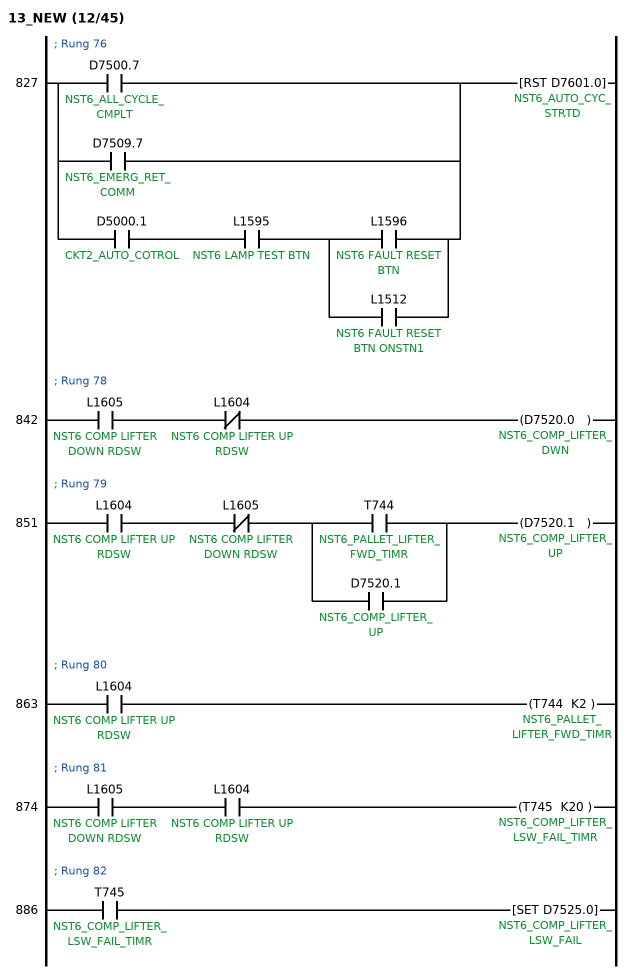
[picture p240: ladder of 13_NEW, rungs at steps 827 to 886]
; Rung 76
827   LD      D7500.7  ; NST6_ALL_CYCLE_CMPLT
      OR      D7509.7  ; NST6_EMERG_RET_COMM
      LD      D5000.1  ; CKT2_AUTO_COTROL
      AND     L1595  ; NST6 LAMP TEST BTN
      LD      L1596  ; NST6 FAULT RESET BTN
      OR      L1512  ; NST6 FAULT RESET BTN ONSTN1
      ANB
      ORB
      RST     D7601.0  ; NST6_AUTO_CYC_STRTD
; Rung 78
842   LD      L1605  ; NST6 COMP LIFTER DOWN RDSW
      ANI     L1604  ; NST6 COMP LIFTER UP RDSW
      OUT     D7520.0  ; NST6_COMP_LIFTER_DWN
; Rung 79
851   LD      L1604  ; NST6 COMP LIFTER UP RDSW
      ANI     L1605  ; NST6 COMP LIFTER DOWN RDSW
      LD      T744  ; NST6_PALLET_LIFTER_FWD_TIMR
      OR      D7520.1  ; NST6_COMP_LIFTER_UP
      ANB
      OUT     D7520.1  ; NST6_COMP_LIFTER_UP
; Rung 80
863   LD      L1604  ; NST6 COMP LIFTER UP RDSW
      OUT     T744 K2  ; NST6_PALLET_LIFTER_FWD_TIMR
; Rung 81
874   LD      L1605  ; NST6 COMP LIFTER DOWN RDSW
      AND     L1604  ; NST6 COMP LIFTER UP RDSW
      OUT     T745 K20  ; NST6_COMP_LIFTER_LSW_FAIL_TIMR
; Rung 82
886   LD      T745  ; NST6_COMP_LIFTER_LSW_FAIL_TIMR
      SET     D7525.0  ; NST6_COMP_LIFTER_LSW_FAIL
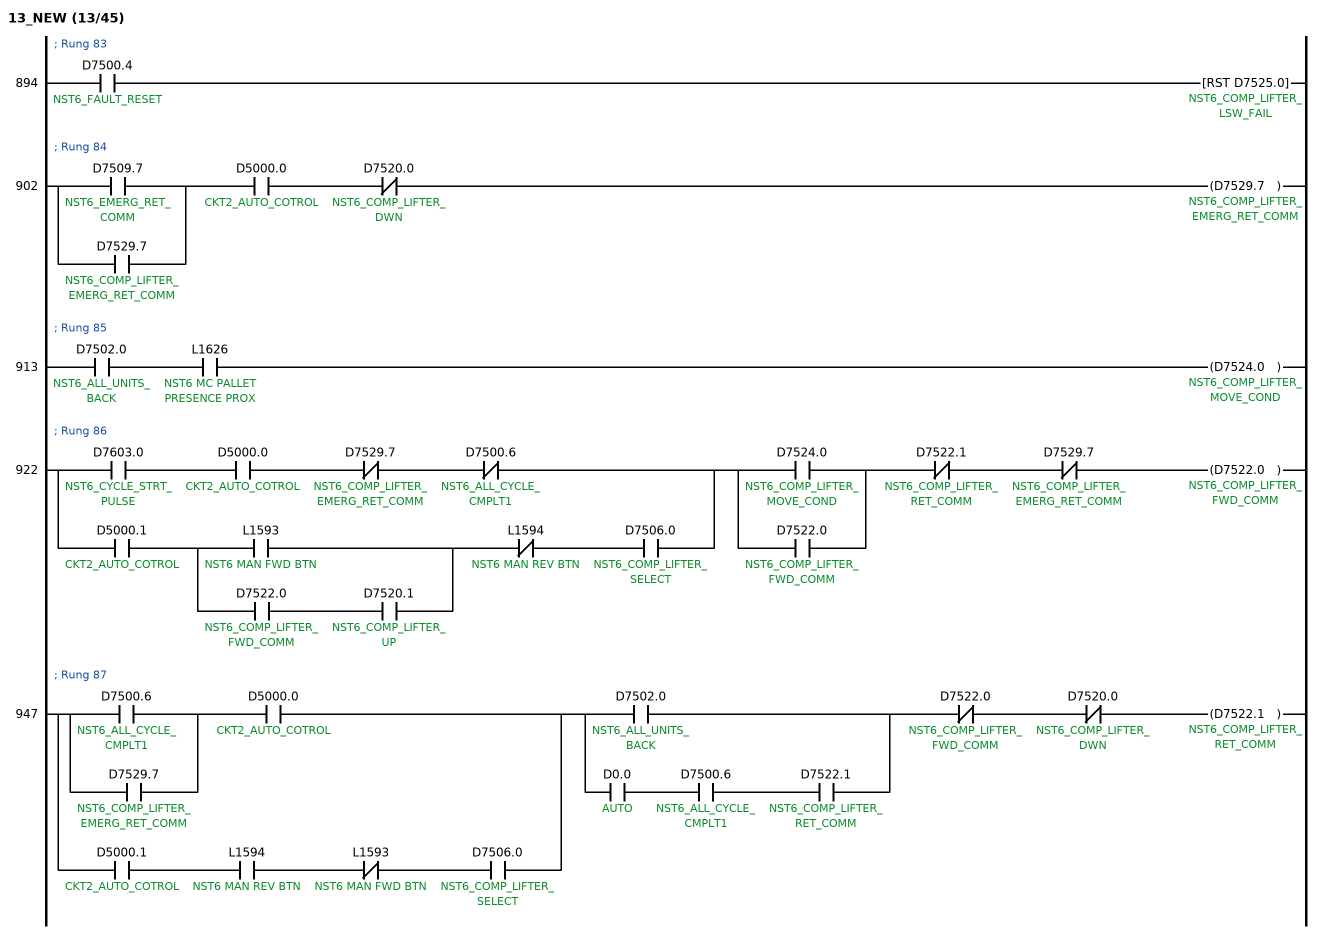
; Rung 83
894   LD      D7500.4  ; NST6_FAULT_RESET
      RST     D7525.0  ; NST6_COMP_LIFTER_LSW_FAIL
; Rung 84
902   LD      D7509.7  ; NST6_EMERG_RET_COMM
      OR      D7529.7  ; NST6_COMP_LIFTER_EMERG_RET_COMM
      AND     D5000.0  ; CKT2_AUTO_COTROL
      ANI     D7520.0  ; NST6_COMP_LIFTER_DWN
      OUT     D7529.7  ; NST6_COMP_LIFTER_EMERG_RET_COMM
; Rung 85
913   LD      D7502.0  ; NST6_ALL_UNITS_BACK
      AND     L1626  ; NST6 MC PALLET PRESENCE PROX
      OUT     D7524.0  ; NST6_COMP_LIFTER_MOVE_COND
; Rung 86
922   LD      D7603.0  ; NST6_CYCLE_STRT_PULSE
      AND     D5000.0  ; CKT2_AUTO_COTROL
      ANI     D7529.7  ; NST6_COMP_LIFTER_EMERG_RET_COMM
      ANI     D7500.6  ; NST6_ALL_CYCLE_CMPLT1
      LD      D5000.1  ; CKT2_AUTO_COTROL
      LD      L1593  ; NST6 MAN FWD BTN
      LD      D7522.0  ; NST6_COMP_LIFTER_FWD_COMM
      AND     D7520.1  ; NST6_COMP_LIFTER_UP
      ORB
      ANB
      ANI     L1594  ; NST6 MAN REV BTN
      AND     D7506.0  ; NST6_COMP_LIFTER_SELECT
      ORB
      LD      D7524.0  ; NST6_COMP_LIFTER_MOVE_COND
      OR      D7522.0  ; NST6_COMP_LIFTER_FWD_COMM
      ANB
      ANI     D7522.1  ; NST6_COMP_LIFTER_RET_COMM
      ANI     D7529.7  ; NST6_COMP_LIFTER_EMERG_RET_COMM
      OUT     D7522.0  ; NST6_COMP_LIFTER_FWD_COMM
; Rung 87
947   LD      D7500.6  ; NST6_ALL_CYCLE_CMPLT1
      OR      D7529.7  ; NST6_COMP_LIFTER_EMERG_RET_COMM
      AND     D5000.0  ; CKT2_AUTO_COTROL
      LD      D5000.1  ; CKT2_AUTO_COTROL
      AND     L1594  ; NST6 MAN REV BTN
      ANI     L1593  ; NST6 MAN FWD BTN
      AND     D7506.0  ; NST6_COMP_LIFTER_SELECT
      ORB
      LD      D7502.0  ; NST6_ALL_UNITS_BACK
      LD      D0.0  ; AUTO
      AND     D7500.6  ; NST6_ALL_CYCLE_CMPLT1
      AND     D7522.1  ; NST6_COMP_LIFTER_RET_COMM
      ORB
      ANB
      ANI     D7522.0  ; NST6_COMP_LIFTER_FWD_COMM
      ANI     D7520.0  ; NST6_COMP_LIFTER_DWN
      OUT     D7522.1  ; NST6_COMP_LIFTER_RET_COMM
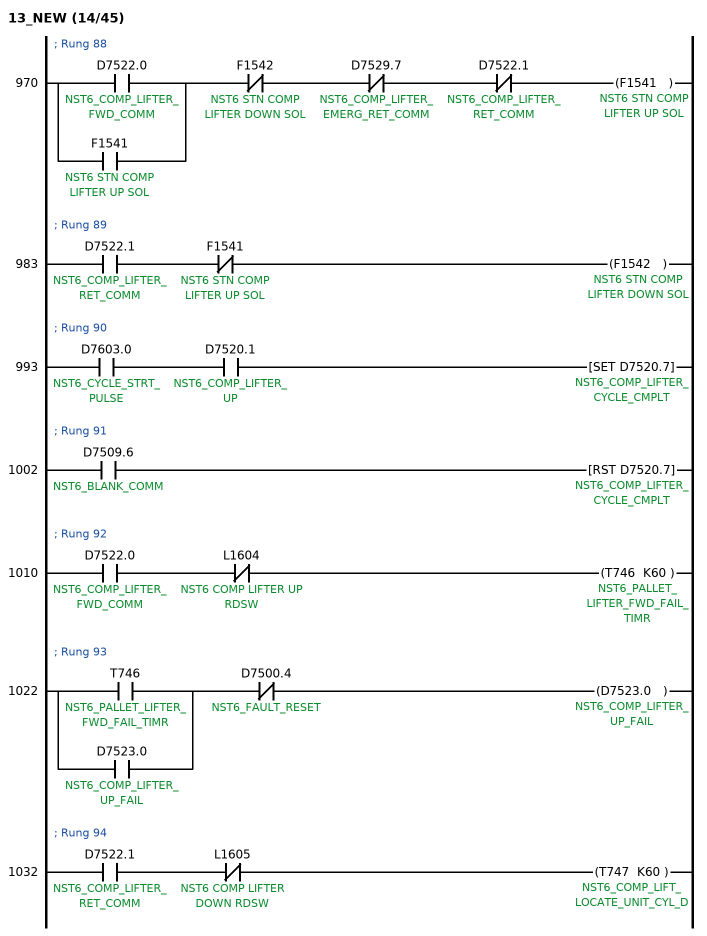
; Rung 88
970   LD      D7522.0  ; NST6_COMP_LIFTER_FWD_COMM
      OR      F1541  ; NST6 STN COMP LIFTER UP SOL
      ANI     F1542  ; NST6 STN COMP LIFTER DOWN SOL
      ANI     D7529.7  ; NST6_COMP_LIFTER_EMERG_RET_COMM
      ANI     D7522.1  ; NST6_COMP_LIFTER_RET_COMM
      OUT     F1541  ; NST6 STN COMP LIFTER UP SOL
; Rung 89
983   LD      D7522.1  ; NST6_COMP_LIFTER_RET_COMM
      ANI     F1541  ; NST6 STN COMP LIFTER UP SOL
      OUT     F1542  ; NST6 STN COMP LIFTER DOWN SOL
; Rung 90
993   LD      D7603.0  ; NST6_CYCLE_STRT_PULSE
      AND     D7520.1  ; NST6_COMP_LIFTER_UP
      SET     D7520.7  ; NST6_COMP_LIFTER_CYCLE_CMPLT
; Rung 91
1002  LD      D7509.6  ; NST6_BLANK_COMM
      RST     D7520.7  ; NST6_COMP_LIFTER_CYCLE_CMPLT
; Rung 92
1010  LD      D7522.0  ; NST6_COMP_LIFTER_FWD_COMM
      ANI     L1604  ; NST6 COMP LIFTER UP RDSW
      OUT     T746 K60  ; NST6_PALLET_LIFTER_FWD_FAIL_TIMR
; Rung 93
1022  LD      T746  ; NST6_PALLET_LIFTER_FWD_FAIL_TIMR
      OR      D7523.0  ; NST6_COMP_LIFTER_UP_FAIL
      ANI     D7500.4  ; NST6_FAULT_RESET
      OUT     D7523.0  ; NST6_COMP_LIFTER_UP_FAIL
; Rung 94
1032  LD      D7522.1  ; NST6_COMP_LIFTER_RET_COMM
      ANI     L1605  ; NST6 COMP LIFTER DOWN RDSW
      OUT     T747 K60  ; NST6_COMP_LIFT_LOCATE_UNIT_CYL_D
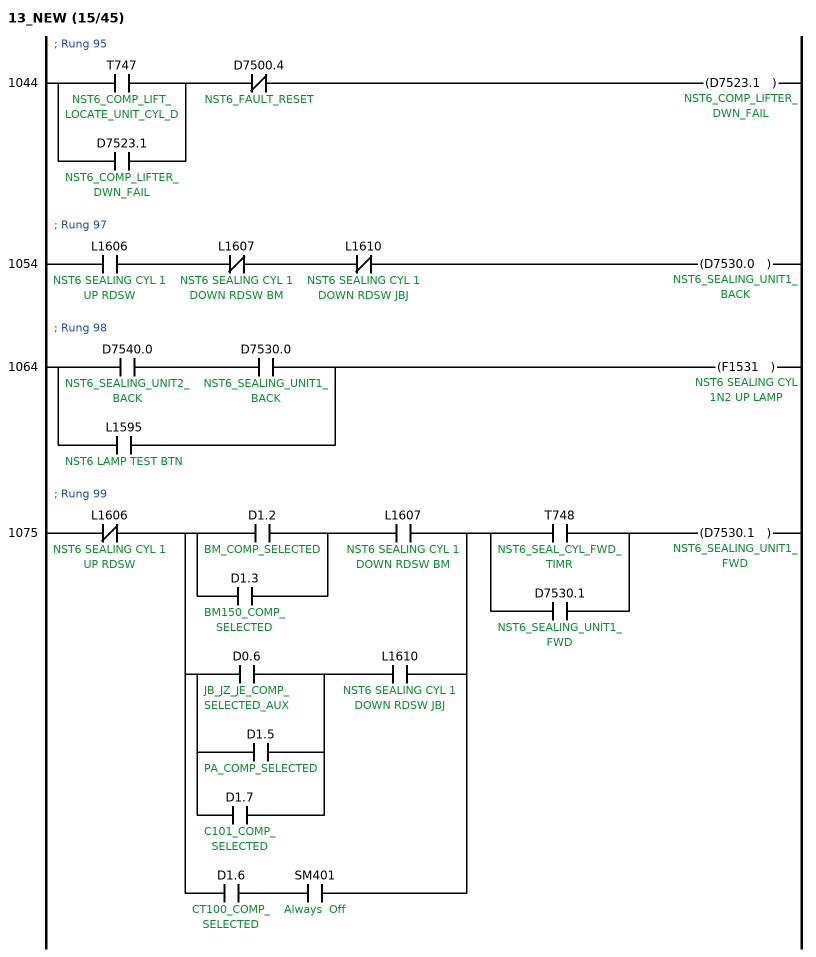
; Rung 95
1044  LD      T747  ; NST6_COMP_LIFT_LOCATE_UNIT_CYL_D
      OR      D7523.1  ; NST6_COMP_LIFTER_DWN_FAIL
      ANI     D7500.4  ; NST6_FAULT_RESET
      OUT     D7523.1  ; NST6_COMP_LIFTER_DWN_FAIL
; Rung 97
1054  LD      L1606  ; NST6 SEALING CYL 1 UP RDSW
      ANI     L1607  ; NST6 SEALING CYL 1 DOWN RDSW BM
      ANI     L1610  ; NST6 SEALING CYL 1 DOWN RDSW JBJ
      OUT     D7530.0  ; NST6_SEALING_UNIT1_BACK
; Rung 98
1064  LD      D7540.0  ; NST6_SEALING_UNIT2_BACK
      AND     D7530.0  ; NST6_SEALING_UNIT1_BACK
      OR      L1595  ; NST6 LAMP TEST BTN
      OUT     F1531  ; NST6 SEALING CYL 1N2 UP LAMP
; Rung 99
1075  LDI     L1606  ; NST6 SEALING CYL 1 UP RDSW
      LD      D1.2  ; BM_COMP_SELECTED
      OR      D1.3  ; BM150_COMP_SELECTED
      AND     L1607  ; NST6 SEALING CYL 1 DOWN RDSW BM
      LD      D0.6  ; JB_JZ_JE_COMP_SELECTED_AUX
      OR      D1.5  ; PA_COMP_SELECTED
      OR      D1.7  ; C101_COMP_SELECTED
      AND     L1610  ; NST6 SEALING CYL 1 DOWN RDSW JBJ
      ORB
      LD      D1.6  ; CT100_COMP_SELECTED
      AND     SM401  ; Always  Off
      ORB
      ANB
      LD      T748  ; NST6_SEAL_CYL_FWD_TIMR
      OR      D7530.1  ; NST6_SEALING_UNIT1_FWD
      ANB
      OUT     D7530.1  ; NST6_SEALING_UNIT1_FWD
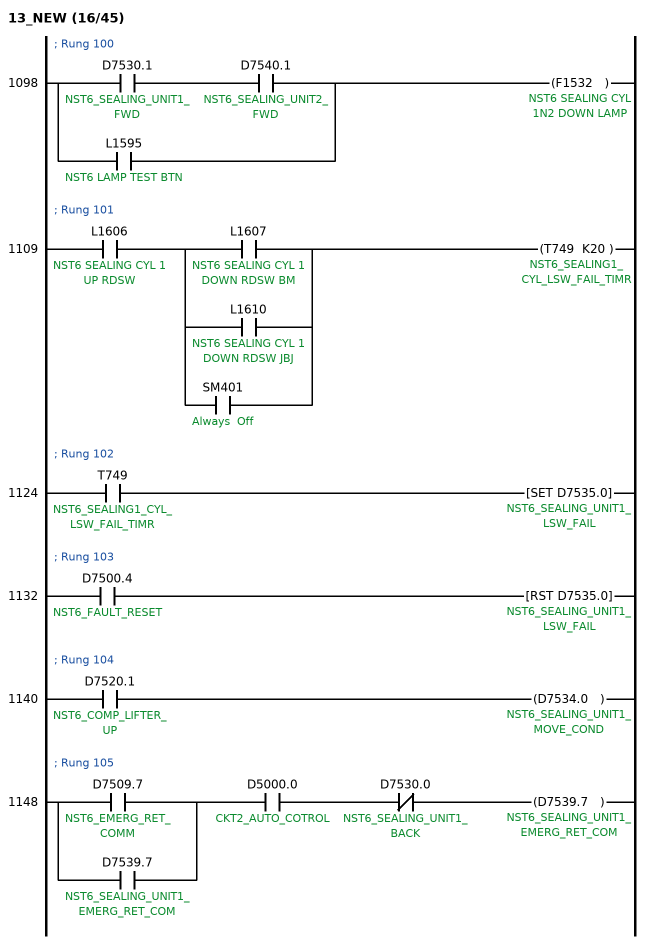
; Rung 100
1098  LD      D7530.1  ; NST6_SEALING_UNIT1_FWD
      AND     D7540.1  ; NST6_SEALING_UNIT2_FWD
      OR      L1595  ; NST6 LAMP TEST BTN
      OUT     F1532  ; NST6 SEALING CYL 1N2 DOWN LAMP
; Rung 101
1109  LD      L1606  ; NST6 SEALING CYL 1 UP RDSW
      LD      L1607  ; NST6 SEALING CYL 1 DOWN RDSW BM
      OR      L1610  ; NST6 SEALING CYL 1 DOWN RDSW JBJ
      OR      SM401  ; Always  Off
      ANB
      OUT     T749 K20  ; NST6_SEALING1_CYL_LSW_FAIL_TIMR
; Rung 102
1124  LD      T749  ; NST6_SEALING1_CYL_LSW_FAIL_TIMR
      SET     D7535.0  ; NST6_SEALING_UNIT1_LSW_FAIL
; Rung 103
1132  LD      D7500.4  ; NST6_FAULT_RESET
      RST     D7535.0  ; NST6_SEALING_UNIT1_LSW_FAIL
; Rung 104
1140  LD      D7520.1  ; NST6_COMP_LIFTER_UP
      OUT     D7534.0  ; NST6_SEALING_UNIT1_MOVE_COND
; Rung 105
1148  LD      D7509.7  ; NST6_EMERG_RET_COMM
      OR      D7539.7  ; NST6_SEALING_UNIT1_EMERG_RET_COM
      AND     D5000.0  ; CKT2_AUTO_COTROL
      ANI     D7530.0  ; NST6_SEALING_UNIT1_BACK
      OUT     D7539.7  ; NST6_SEALING_UNIT1_EMERG_RET_COM
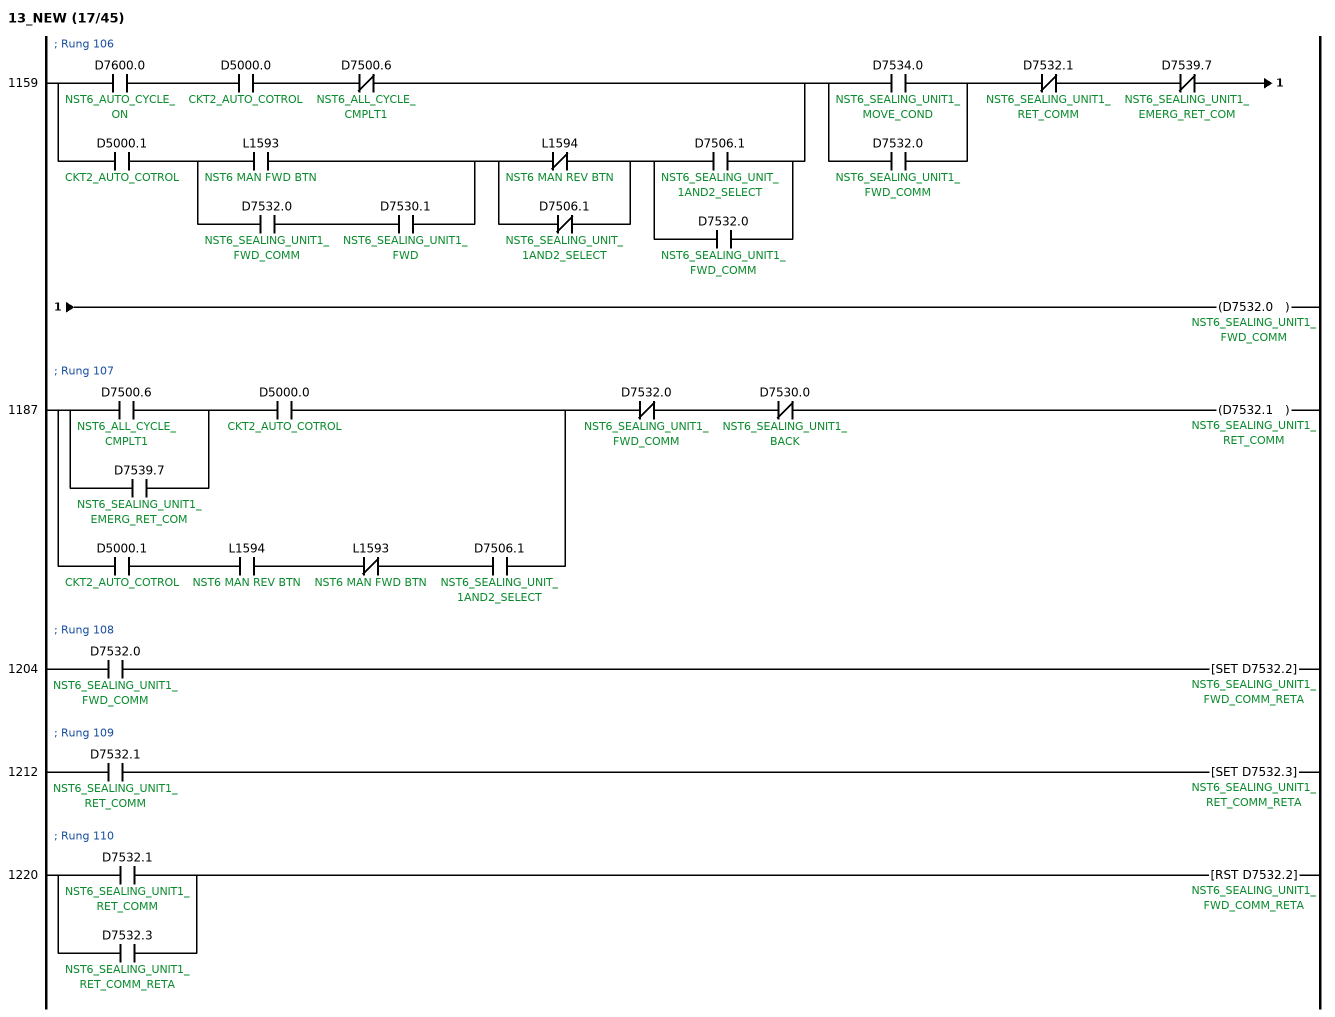
; Rung 106
1159  LD      D7600.0  ; NST6_AUTO_CYCLE_ON
      AND     D5000.0  ; CKT2_AUTO_COTROL
      ANI     D7500.6  ; NST6_ALL_CYCLE_CMPLT1
      LD      D5000.1  ; CKT2_AUTO_COTROL
      LD      L1593  ; NST6 MAN FWD BTN
      LD      D7532.0  ; NST6_SEALING_UNIT1_FWD_COMM
      AND     D7530.1  ; NST6_SEALING_UNIT1_FWD
      ORB
      ANB
      LDI     L1594  ; NST6 MAN REV BTN
      ORI     D7506.1  ; NST6_SEALING_UNIT_1AND2_SELECT
      ANB
      LD      D7506.1  ; NST6_SEALING_UNIT_1AND2_SELECT
      OR      D7532.0  ; NST6_SEALING_UNIT1_FWD_COMM
      ANB
      ORB
      LD      D7534.0  ; NST6_SEALING_UNIT1_MOVE_COND
      OR      D7532.0  ; NST6_SEALING_UNIT1_FWD_COMM
      ANB
      ANI     D7532.1  ; NST6_SEALING_UNIT1_RET_COMM
      ANI     D7539.7  ; NST6_SEALING_UNIT1_EMERG_RET_COM
      OUT     D7532.0  ; NST6_SEALING_UNIT1_FWD_COMM
; Rung 107
1187  LD      D7500.6  ; NST6_ALL_CYCLE_CMPLT1
      OR      D7539.7  ; NST6_SEALING_UNIT1_EMERG_RET_COM
      AND     D5000.0  ; CKT2_AUTO_COTROL
      LD      D5000.1  ; CKT2_AUTO_COTROL
      AND     L1594  ; NST6 MAN REV BTN
      ANI     L1593  ; NST6 MAN FWD BTN
      AND     D7506.1  ; NST6_SEALING_UNIT_1AND2_SELECT
      ORB
      ANI     D7532.0  ; NST6_SEALING_UNIT1_FWD_COMM
      ANI     D7530.0  ; NST6_SEALING_UNIT1_BACK
      OUT     D7532.1  ; NST6_SEALING_UNIT1_RET_COMM
; Rung 108
1204  LD      D7532.0  ; NST6_SEALING_UNIT1_FWD_COMM
      SET     D7532.2  ; NST6_SEALING_UNIT1_FWD_COMM_RETA
; Rung 109
1212  LD      D7532.1  ; NST6_SEALING_UNIT1_RET_COMM
      SET     D7532.3  ; NST6_SEALING_UNIT1_RET_COMM_RETA
; Rung 110
1220  LD      D7532.1  ; NST6_SEALING_UNIT1_RET_COMM
      OR      D7532.3  ; NST6_SEALING_UNIT1_RET_COMM_RETA
      RST     D7532.2  ; NST6_SEALING_UNIT1_FWD_COMM_RETA
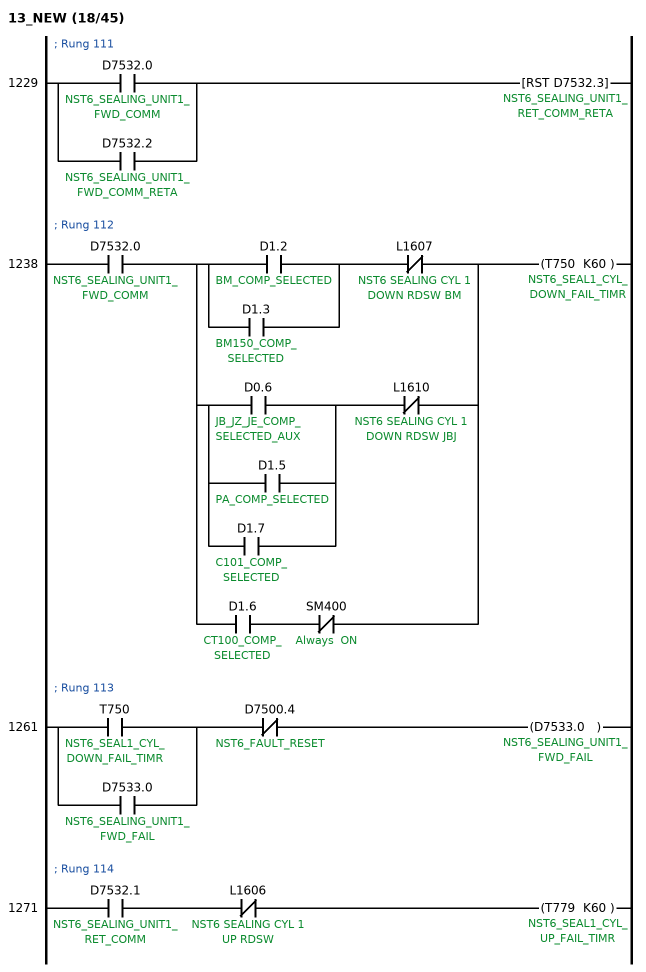
; Rung 111
1229  LD      D7532.0  ; NST6_SEALING_UNIT1_FWD_COMM
      OR      D7532.2  ; NST6_SEALING_UNIT1_FWD_COMM_RETA
      RST     D7532.3  ; NST6_SEALING_UNIT1_RET_COMM_RETA
; Rung 112
1238  LD      D7532.0  ; NST6_SEALING_UNIT1_FWD_COMM
      LD      D1.2  ; BM_COMP_SELECTED
      OR      D1.3  ; BM150_COMP_SELECTED
      ANI     L1607  ; NST6 SEALING CYL 1 DOWN RDSW BM
      LD      D0.6  ; JB_JZ_JE_COMP_SELECTED_AUX
      OR      D1.5  ; PA_COMP_SELECTED
      OR      D1.7  ; C101_COMP_SELECTED
      ANI     L1610  ; NST6 SEALING CYL 1 DOWN RDSW JBJ
      ORB
      LD      D1.6  ; CT100_COMP_SELECTED
      ANI     SM400  ; Always  ON
      ORB
      ANB
      OUT     T750 K60  ; NST6_SEAL1_CYL_DOWN_FAIL_TIMR
; Rung 113
1261  LD      T750  ; NST6_SEAL1_CYL_DOWN_FAIL_TIMR
      OR      D7533.0  ; NST6_SEALING_UNIT1_FWD_FAIL
      ANI     D7500.4  ; NST6_FAULT_RESET
      OUT     D7533.0  ; NST6_SEALING_UNIT1_FWD_FAIL
; Rung 114
1271  LD      D7532.1  ; NST6_SEALING_UNIT1_RET_COMM
      ANI     L1606  ; NST6 SEALING CYL 1 UP RDSW
      OUT     T779 K60  ; NST6_SEAL1_CYL_UP_FAIL_TIMR
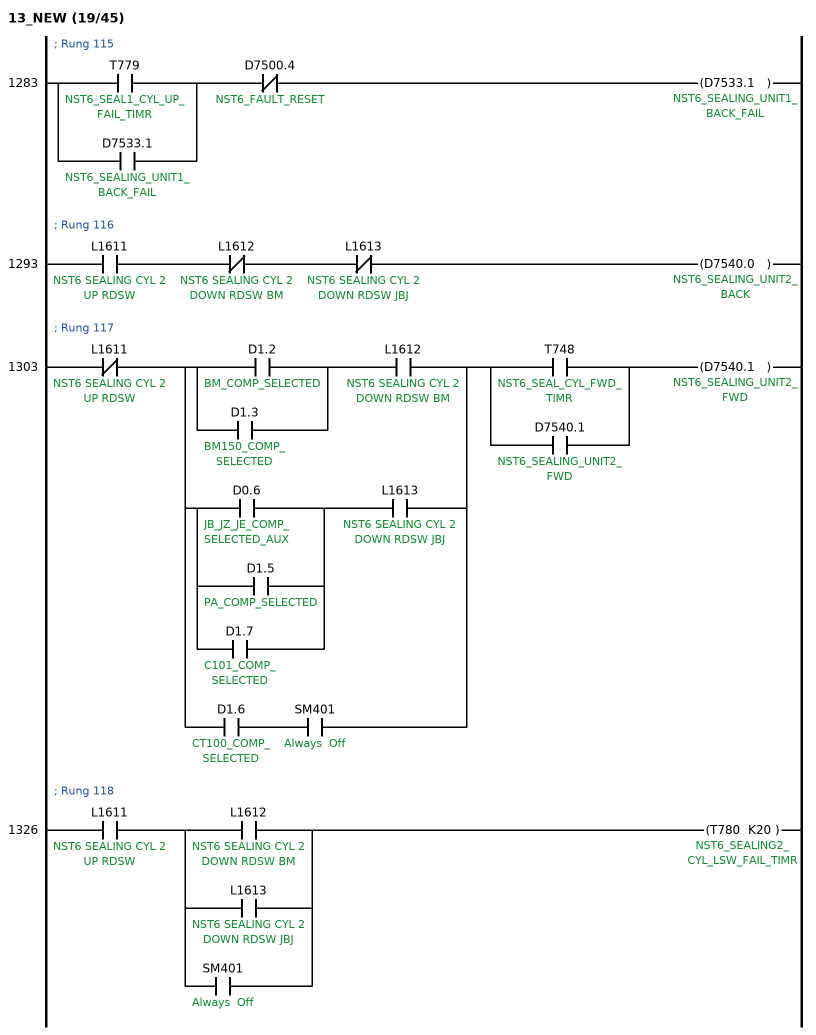
; Rung 115
1283  LD      T779  ; NST6_SEAL1_CYL_UP_FAIL_TIMR
      OR      D7533.1  ; NST6_SEALING_UNIT1_BACK_FAIL
      ANI     D7500.4  ; NST6_FAULT_RESET
      OUT     D7533.1  ; NST6_SEALING_UNIT1_BACK_FAIL
; Rung 116
1293  LD      L1611  ; NST6 SEALING CYL 2 UP RDSW
      ANI     L1612  ; NST6 SEALING CYL 2 DOWN RDSW BM
      ANI     L1613  ; NST6 SEALING CYL 2 DOWN RDSW JBJ
      OUT     D7540.0  ; NST6_SEALING_UNIT2_BACK
; Rung 117
1303  LDI     L1611  ; NST6 SEALING CYL 2 UP RDSW
      LD      D1.2  ; BM_COMP_SELECTED
      OR      D1.3  ; BM150_COMP_SELECTED
      AND     L1612  ; NST6 SEALING CYL 2 DOWN RDSW BM
      LD      D0.6  ; JB_JZ_JE_COMP_SELECTED_AUX
      OR      D1.5  ; PA_COMP_SELECTED
      OR      D1.7  ; C101_COMP_SELECTED
      AND     L1613  ; NST6 SEALING CYL 2 DOWN RDSW JBJ
      ORB
      LD      D1.6  ; CT100_COMP_SELECTED
      AND     SM401  ; Always  Off
      ORB
      ANB
      LD      T748  ; NST6_SEAL_CYL_FWD_TIMR
      OR      D7540.1  ; NST6_SEALING_UNIT2_FWD
      ANB
      OUT     D7540.1  ; NST6_SEALING_UNIT2_FWD
; Rung 118
1326  LD      L1611  ; NST6 SEALING CYL 2 UP RDSW
      LD      L1612  ; NST6 SEALING CYL 2 DOWN RDSW BM
      OR      L1613  ; NST6 SEALING CYL 2 DOWN RDSW JBJ
      OR      SM401  ; Always  Off
      ANB
      OUT     T780 K20  ; NST6_SEALING2_CYL_LSW_FAIL_TIMR
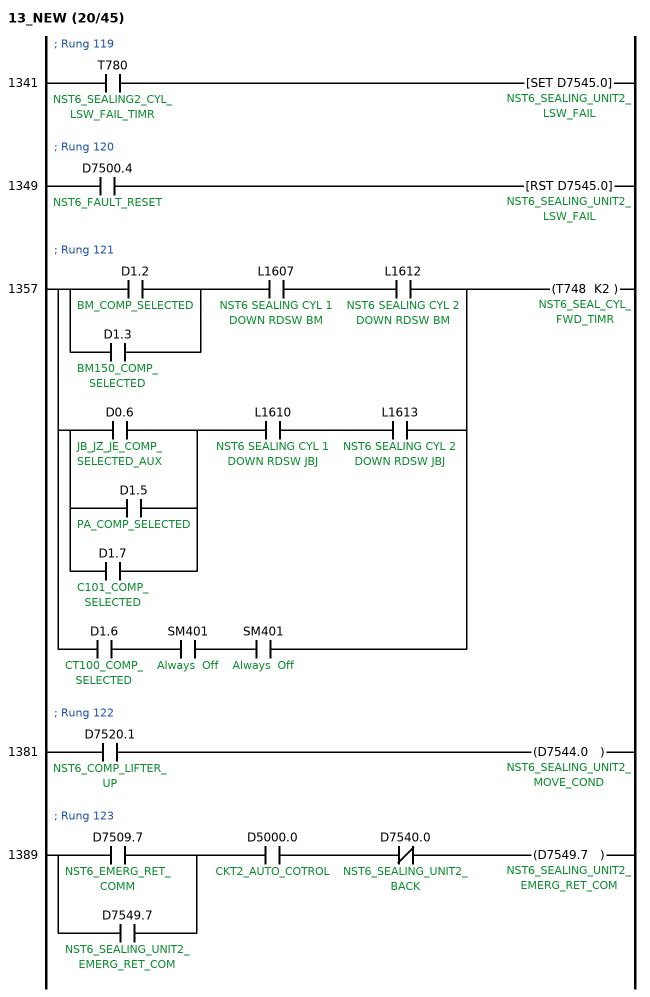
; Rung 119
1341  LD      T780  ; NST6_SEALING2_CYL_LSW_FAIL_TIMR
      SET     D7545.0  ; NST6_SEALING_UNIT2_LSW_FAIL
; Rung 120
1349  LD      D7500.4  ; NST6_FAULT_RESET
      RST     D7545.0  ; NST6_SEALING_UNIT2_LSW_FAIL
; Rung 121
1357  LD      D1.2  ; BM_COMP_SELECTED
      OR      D1.3  ; BM150_COMP_SELECTED
      AND     L1607  ; NST6 SEALING CYL 1 DOWN RDSW BM
      AND     L1612  ; NST6 SEALING CYL 2 DOWN RDSW BM
      LD      D0.6  ; JB_JZ_JE_COMP_SELECTED_AUX
      OR      D1.5  ; PA_COMP_SELECTED
      OR      D1.7  ; C101_COMP_SELECTED
      AND     L1610  ; NST6 SEALING CYL 1 DOWN RDSW JBJ
      AND     L1613  ; NST6 SEALING CYL 2 DOWN RDSW JBJ
      ORB
      LD      D1.6  ; CT100_COMP_SELECTED
      AND     SM401  ; Always  Off
      AND     SM401  ; Always  Off
      ORB
      OUT     T748 K2  ; NST6_SEAL_CYL_FWD_TIMR
; Rung 122
1381  LD      D7520.1  ; NST6_COMP_LIFTER_UP
      OUT     D7544.0  ; NST6_SEALING_UNIT2_MOVE_COND
; Rung 123
1389  LD      D7509.7  ; NST6_EMERG_RET_COMM
      OR      D7549.7  ; NST6_SEALING_UNIT2_EMERG_RET_COM
      AND     D5000.0  ; CKT2_AUTO_COTROL
      ANI     D7540.0  ; NST6_SEALING_UNIT2_BACK
      OUT     D7549.7  ; NST6_SEALING_UNIT2_EMERG_RET_COM
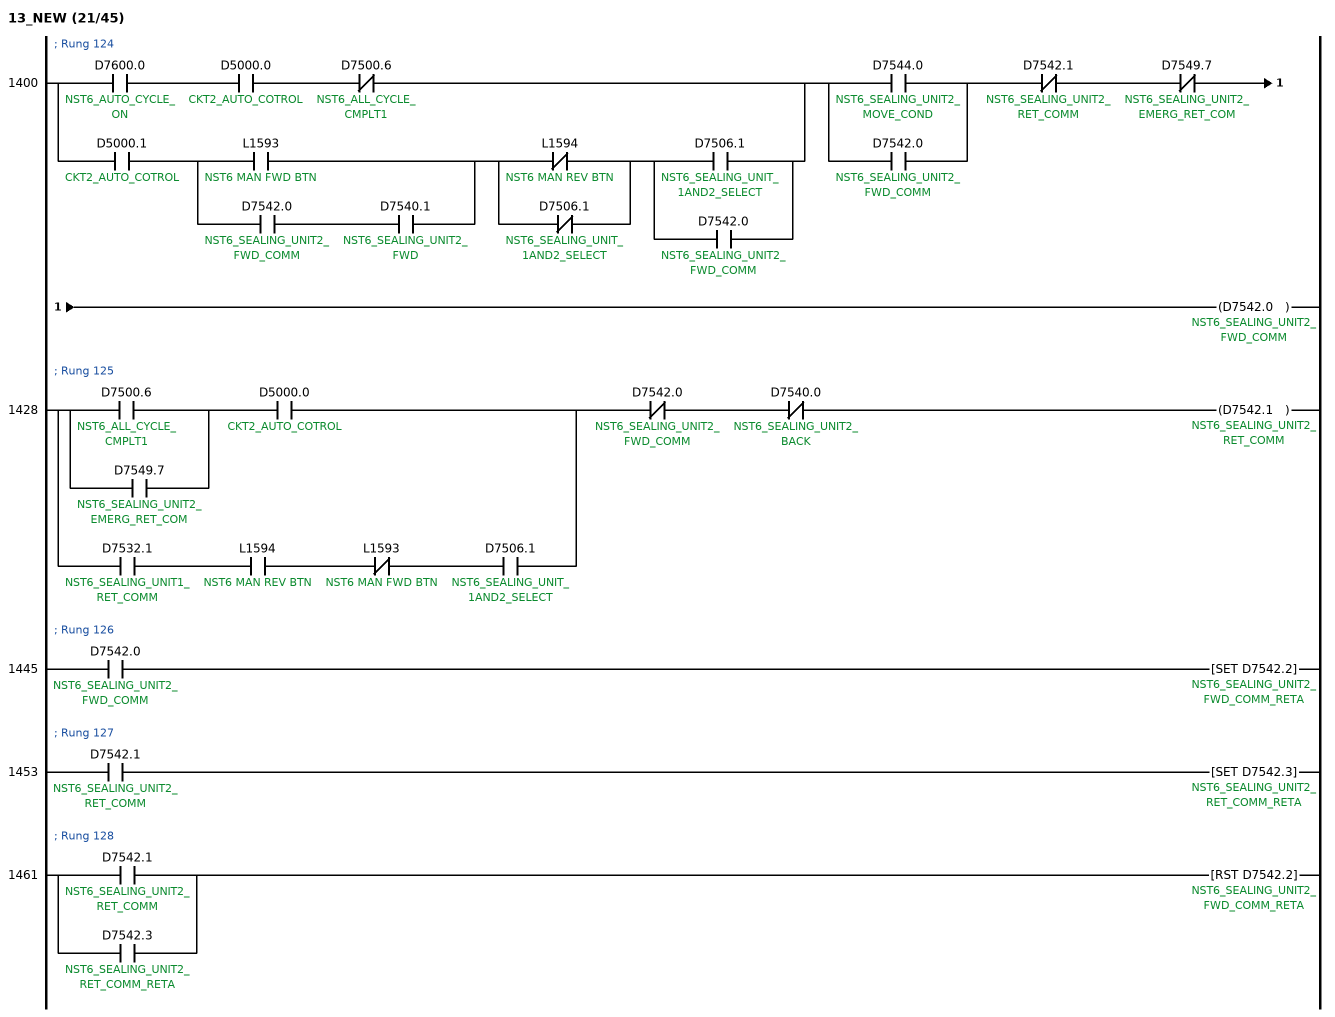
; Rung 124
1400  LD      D7600.0  ; NST6_AUTO_CYCLE_ON
      AND     D5000.0  ; CKT2_AUTO_COTROL
      ANI     D7500.6  ; NST6_ALL_CYCLE_CMPLT1
      LD      D5000.1  ; CKT2_AUTO_COTROL
      LD      L1593  ; NST6 MAN FWD BTN
      LD      D7542.0  ; NST6_SEALING_UNIT2_FWD_COMM
      AND     D7540.1  ; NST6_SEALING_UNIT2_FWD
      ORB
      ANB
      LDI     L1594  ; NST6 MAN REV BTN
      ORI     D7506.1  ; NST6_SEALING_UNIT_1AND2_SELECT
      ANB
      LD      D7506.1  ; NST6_SEALING_UNIT_1AND2_SELECT
      OR      D7542.0  ; NST6_SEALING_UNIT2_FWD_COMM
      ANB
      ORB
      LD      D7544.0  ; NST6_SEALING_UNIT2_MOVE_COND
      OR      D7542.0  ; NST6_SEALING_UNIT2_FWD_COMM
      ANB
      ANI     D7542.1  ; NST6_SEALING_UNIT2_RET_COMM
      ANI     D7549.7  ; NST6_SEALING_UNIT2_EMERG_RET_COM
      OUT     D7542.0  ; NST6_SEALING_UNIT2_FWD_COMM
; Rung 125
1428  LD      D7500.6  ; NST6_ALL_CYCLE_CMPLT1
      OR      D7549.7  ; NST6_SEALING_UNIT2_EMERG_RET_COM
      AND     D5000.0  ; CKT2_AUTO_COTROL
      LD      D7532.1  ; NST6_SEALING_UNIT1_RET_COMM
      AND     L1594  ; NST6 MAN REV BTN
      ANI     L1593  ; NST6 MAN FWD BTN
      AND     D7506.1  ; NST6_SEALING_UNIT_1AND2_SELECT
      ORB
      ANI     D7542.0  ; NST6_SEALING_UNIT2_FWD_COMM
      ANI     D7540.0  ; NST6_SEALING_UNIT2_BACK
      OUT     D7542.1  ; NST6_SEALING_UNIT2_RET_COMM
; Rung 126
1445  LD      D7542.0  ; NST6_SEALING_UNIT2_FWD_COMM
      SET     D7542.2  ; NST6_SEALING_UNIT2_FWD_COMM_RETA
; Rung 127
1453  LD      D7542.1  ; NST6_SEALING_UNIT2_RET_COMM
      SET     D7542.3  ; NST6_SEALING_UNIT2_RET_COMM_RETA
; Rung 128
1461  LD      D7542.1  ; NST6_SEALING_UNIT2_RET_COMM
      OR      D7542.3  ; NST6_SEALING_UNIT2_RET_COMM_RETA
      RST     D7542.2  ; NST6_SEALING_UNIT2_FWD_COMM_RETA
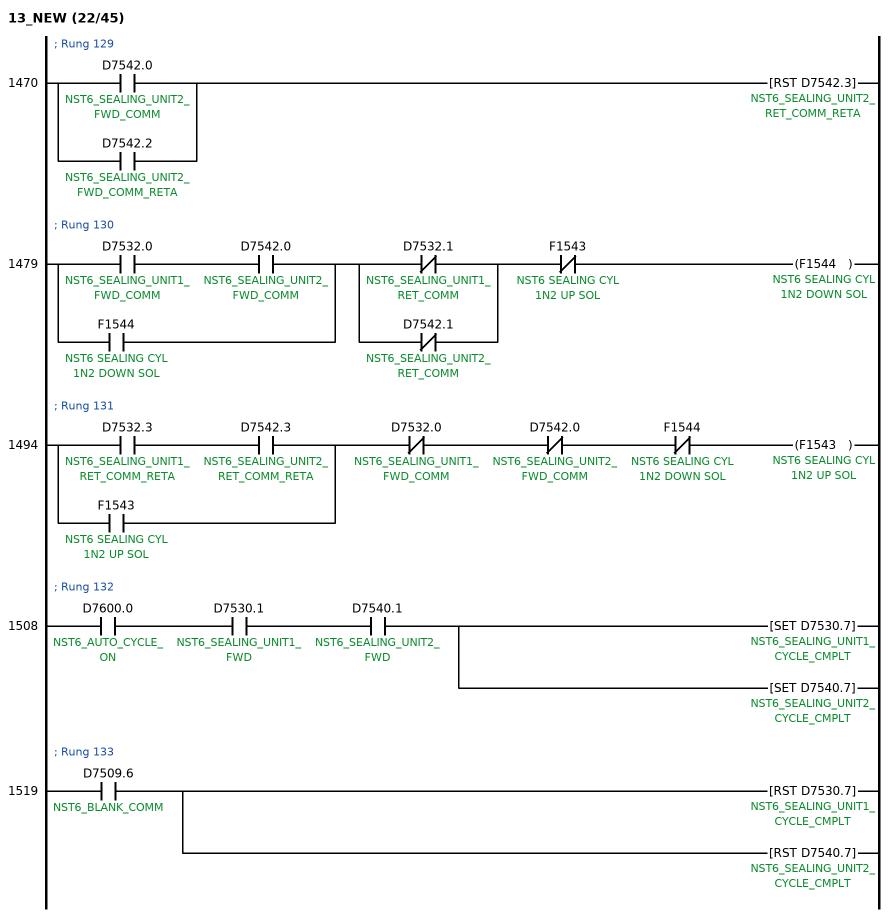
; Rung 129
1470  LD      D7542.0  ; NST6_SEALING_UNIT2_FWD_COMM
      OR      D7542.2  ; NST6_SEALING_UNIT2_FWD_COMM_RETA
      RST     D7542.3  ; NST6_SEALING_UNIT2_RET_COMM_RETA
; Rung 130
1479  LD      D7532.0  ; NST6_SEALING_UNIT1_FWD_COMM
      AND     D7542.0  ; NST6_SEALING_UNIT2_FWD_COMM
      OR      F1544  ; NST6 SEALING CYL 1N2 DOWN SOL
      LDI     D7532.1  ; NST6_SEALING_UNIT1_RET_COMM
      ORI     D7542.1  ; NST6_SEALING_UNIT2_RET_COMM
      ANB
      ANI     F1543  ; NST6 SEALING CYL 1N2 UP SOL
      OUT     F1544  ; NST6 SEALING CYL 1N2 DOWN SOL
; Rung 131
1494  LD      D7532.3  ; NST6_SEALING_UNIT1_RET_COMM_RETA
      AND     D7542.3  ; NST6_SEALING_UNIT2_RET_COMM_RETA
      OR      F1543  ; NST6 SEALING CYL 1N2 UP SOL
      ANI     D7532.0  ; NST6_SEALING_UNIT1_FWD_COMM
      ANI     D7542.0  ; NST6_SEALING_UNIT2_FWD_COMM
      ANI     F1544  ; NST6 SEALING CYL 1N2 DOWN SOL
      OUT     F1543  ; NST6 SEALING CYL 1N2 UP SOL
; Rung 132
1508  LD      D7600.0  ; NST6_AUTO_CYCLE_ON
      AND     D7530.1  ; NST6_SEALING_UNIT1_FWD
      AND     D7540.1  ; NST6_SEALING_UNIT2_FWD
      SET     D7530.7  ; NST6_SEALING_UNIT1_CYCLE_CMPLT
      SET     D7540.7  ; NST6_SEALING_UNIT2_CYCLE_CMPLT
; Rung 133
1519  LD      D7509.6  ; NST6_BLANK_COMM
      RST     D7530.7  ; NST6_SEALING_UNIT1_CYCLE_CMPLT
      RST     D7540.7  ; NST6_SEALING_UNIT2_CYCLE_CMPLT
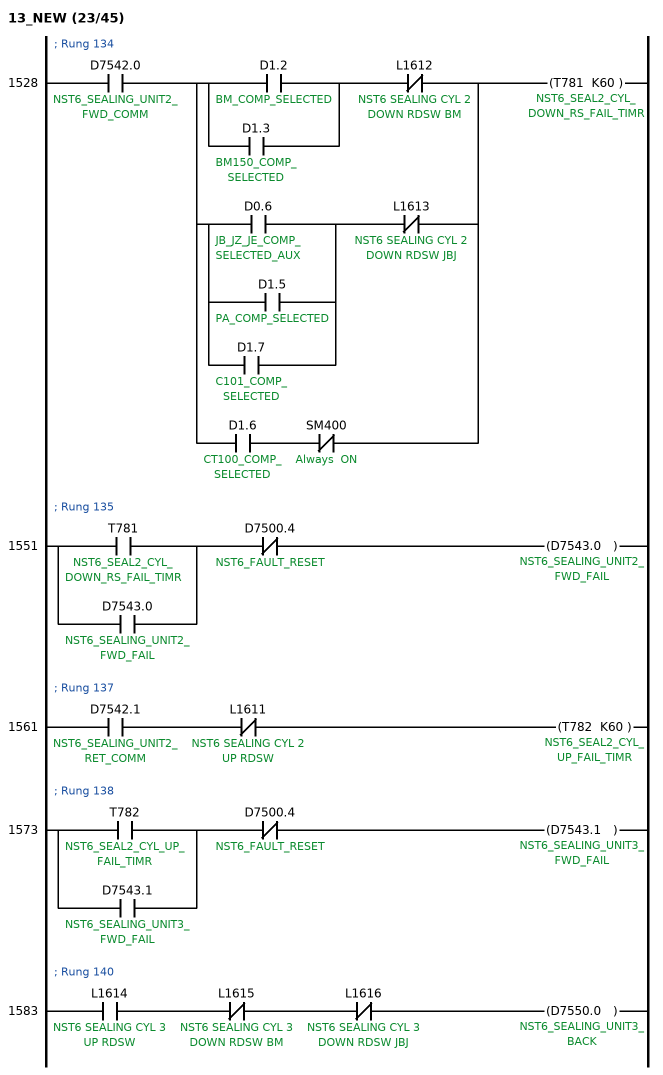
; Rung 134
1528  LD      D7542.0  ; NST6_SEALING_UNIT2_FWD_COMM
      LD      D1.2  ; BM_COMP_SELECTED
      OR      D1.3  ; BM150_COMP_SELECTED
      ANI     L1612  ; NST6 SEALING CYL 2 DOWN RDSW BM
      LD      D0.6  ; JB_JZ_JE_COMP_SELECTED_AUX
      OR      D1.5  ; PA_COMP_SELECTED
      OR      D1.7  ; C101_COMP_SELECTED
      ANI     L1613  ; NST6 SEALING CYL 2 DOWN RDSW JBJ
      ORB
      LD      D1.6  ; CT100_COMP_SELECTED
      ANI     SM400  ; Always  ON
      ORB
      ANB
      OUT     T781 K60  ; NST6_SEAL2_CYL_DOWN_RS_FAIL_TIMR
; Rung 135
1551  LD      T781  ; NST6_SEAL2_CYL_DOWN_RS_FAIL_TIMR
      OR      D7543.0  ; NST6_SEALING_UNIT2_FWD_FAIL
      ANI     D7500.4  ; NST6_FAULT_RESET
      OUT     D7543.0  ; NST6_SEALING_UNIT2_FWD_FAIL
; Rung 137
1561  LD      D7542.1  ; NST6_SEALING_UNIT2_RET_COMM
      ANI     L1611  ; NST6 SEALING CYL 2 UP RDSW
      OUT     T782 K60  ; NST6_SEAL2_CYL_UP_FAIL_TIMR
; Rung 138
1573  LD      T782  ; NST6_SEAL2_CYL_UP_FAIL_TIMR
      OR      D7543.1  ; NST6_SEALING_UNIT3_FWD_FAIL
      ANI     D7500.4  ; NST6_FAULT_RESET
      OUT     D7543.1  ; NST6_SEALING_UNIT3_FWD_FAIL
; Rung 140
1583  LD      L1614  ; NST6 SEALING CYL 3 UP RDSW
      ANI     L1615  ; NST6 SEALING CYL 3 DOWN RDSW BM
      ANI     L1616  ; NST6 SEALING CYL 3 DOWN RDSW JBJ
      OUT     D7550.0  ; NST6_SEALING_UNIT3_BACK
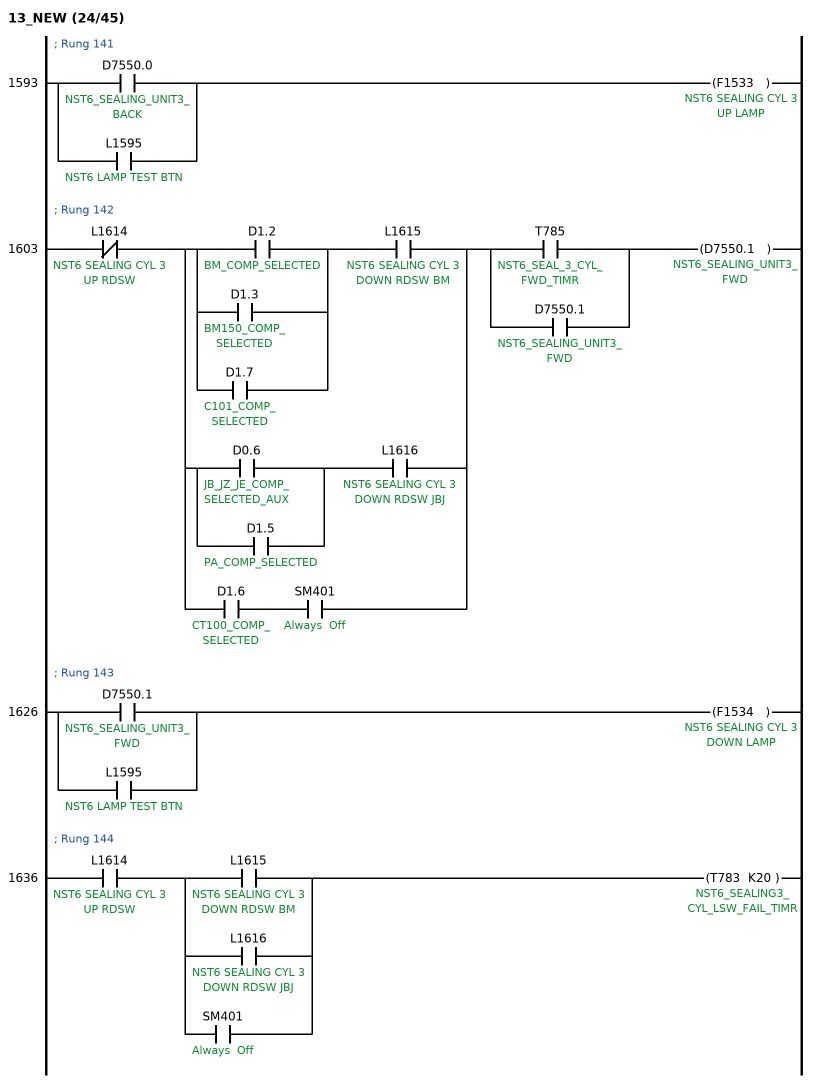
; Rung 141
1593  LD      D7550.0  ; NST6_SEALING_UNIT3_BACK
      OR      L1595  ; NST6 LAMP TEST BTN
      OUT     F1533  ; NST6 SEALING CYL 3 UP LAMP
; Rung 142
1603  LDI     L1614  ; NST6 SEALING CYL 3 UP RDSW
      LD      D1.2  ; BM_COMP_SELECTED
      OR      D1.3  ; BM150_COMP_SELECTED
      OR      D1.7  ; C101_COMP_SELECTED
      AND     L1615  ; NST6 SEALING CYL 3 DOWN RDSW BM
      LD      D0.6  ; JB_JZ_JE_COMP_SELECTED_AUX
      OR      D1.5  ; PA_COMP_SELECTED
      AND     L1616  ; NST6 SEALING CYL 3 DOWN RDSW JBJ
      ORB
      LD      D1.6  ; CT100_COMP_SELECTED
      AND     SM401  ; Always  Off
      ORB
      ANB
      LD      T785  ; NST6_SEAL_3_CYL_FWD_TIMR
      OR      D7550.1  ; NST6_SEALING_UNIT3_FWD
      ANB
      OUT     D7550.1  ; NST6_SEALING_UNIT3_FWD
; Rung 143
1626  LD      D7550.1  ; NST6_SEALING_UNIT3_FWD
      OR      L1595  ; NST6 LAMP TEST BTN
      OUT     F1534  ; NST6 SEALING CYL 3 DOWN LAMP
; Rung 144
1636  LD      L1614  ; NST6 SEALING CYL 3 UP RDSW
      LD      L1615  ; NST6 SEALING CYL 3 DOWN RDSW BM
      OR      L1616  ; NST6 SEALING CYL 3 DOWN RDSW JBJ
      OR      SM401  ; Always  Off
      ANB
      OUT     T783 K20  ; NST6_SEALING3_CYL_LSW_FAIL_TIMR
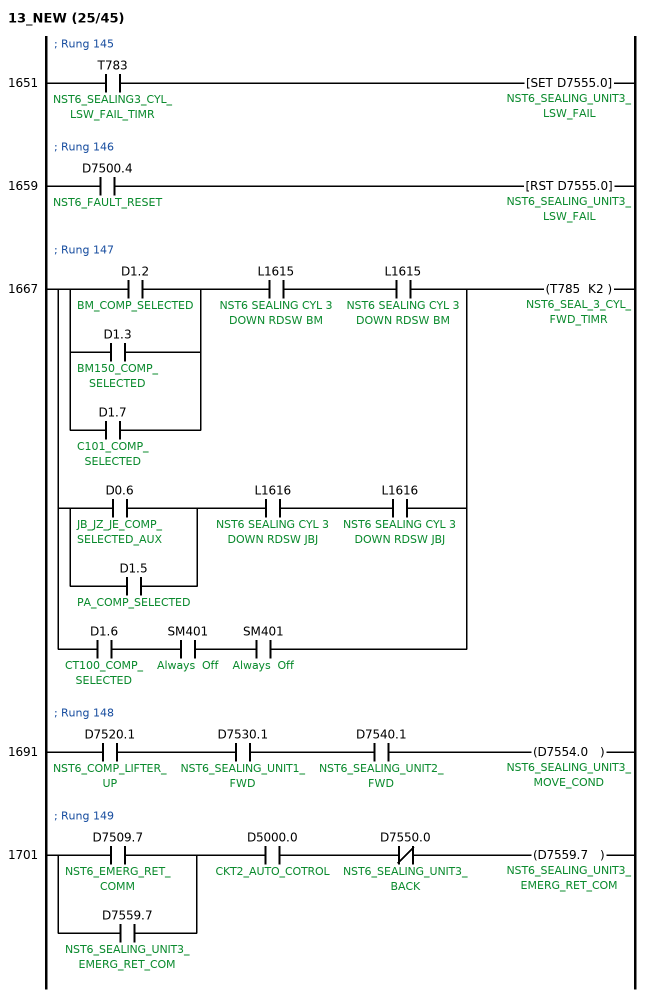
; Rung 145
1651  LD      T783  ; NST6_SEALING3_CYL_LSW_FAIL_TIMR
      SET     D7555.0  ; NST6_SEALING_UNIT3_LSW_FAIL
; Rung 146
1659  LD      D7500.4  ; NST6_FAULT_RESET
      RST     D7555.0  ; NST6_SEALING_UNIT3_LSW_FAIL
; Rung 147
1667  LD      D1.2  ; BM_COMP_SELECTED
      OR      D1.3  ; BM150_COMP_SELECTED
      OR      D1.7  ; C101_COMP_SELECTED
      AND     L1615  ; NST6 SEALING CYL 3 DOWN RDSW BM
      AND     L1615  ; NST6 SEALING CYL 3 DOWN RDSW BM
      LD      D0.6  ; JB_JZ_JE_COMP_SELECTED_AUX
      OR      D1.5  ; PA_COMP_SELECTED
      AND     L1616  ; NST6 SEALING CYL 3 DOWN RDSW JBJ
      AND     L1616  ; NST6 SEALING CYL 3 DOWN RDSW JBJ
      ORB
      LD      D1.6  ; CT100_COMP_SELECTED
      AND     SM401  ; Always  Off
      AND     SM401  ; Always  Off
      ORB
      OUT     T785 K2  ; NST6_SEAL_3_CYL_FWD_TIMR
; Rung 148
1691  LD      D7520.1  ; NST6_COMP_LIFTER_UP
      AND     D7530.1  ; NST6_SEALING_UNIT1_FWD
      AND     D7540.1  ; NST6_SEALING_UNIT2_FWD
      OUT     D7554.0  ; NST6_SEALING_UNIT3_MOVE_COND
; Rung 149
1701  LD      D7509.7  ; NST6_EMERG_RET_COMM
      OR      D7559.7  ; NST6_SEALING_UNIT3_EMERG_RET_COM
      AND     D5000.0  ; CKT2_AUTO_COTROL
      ANI     D7550.0  ; NST6_SEALING_UNIT3_BACK
      OUT     D7559.7  ; NST6_SEALING_UNIT3_EMERG_RET_COM
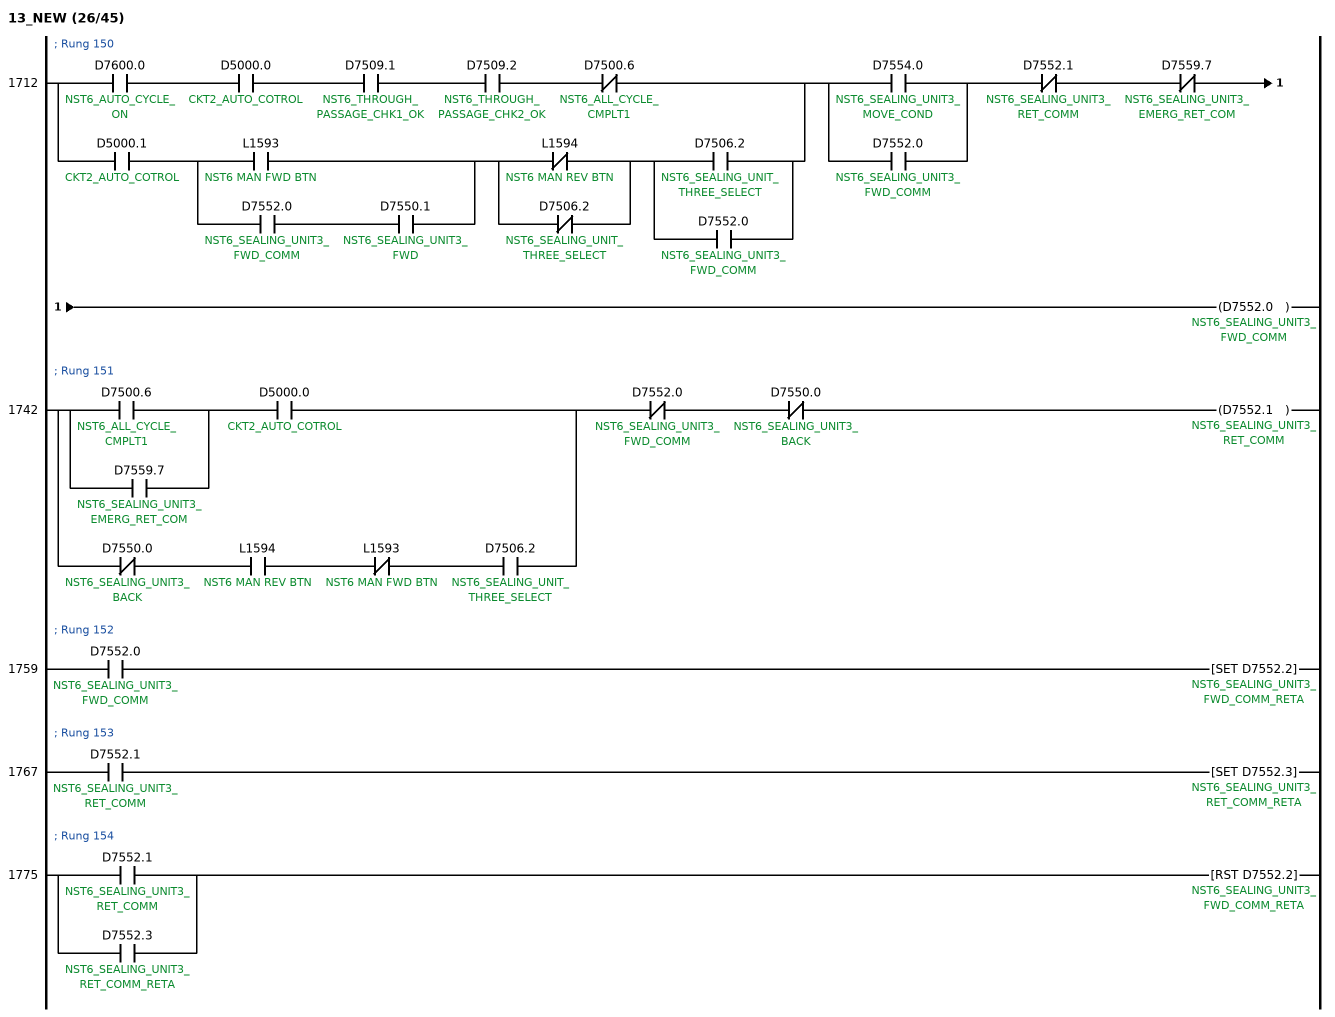
; Rung 150
1712  LD      D7600.0  ; NST6_AUTO_CYCLE_ON
      AND     D5000.0  ; CKT2_AUTO_COTROL
      AND     D7509.1  ; NST6_THROUGH_PASSAGE_CHK1_OK
      AND     D7509.2  ; NST6_THROUGH_PASSAGE_CHK2_OK
      ANI     D7500.6  ; NST6_ALL_CYCLE_CMPLT1
      LD      D5000.1  ; CKT2_AUTO_COTROL
      LD      L1593  ; NST6 MAN FWD BTN
      LD      D7552.0  ; NST6_SEALING_UNIT3_FWD_COMM
      AND     D7550.1  ; NST6_SEALING_UNIT3_FWD
      ORB
      ANB
      LDI     L1594  ; NST6 MAN REV BTN
      ORI     D7506.2  ; NST6_SEALING_UNIT_THREE_SELECT
      ANB
      LD      D7506.2  ; NST6_SEALING_UNIT_THREE_SELECT
      OR      D7552.0  ; NST6_SEALING_UNIT3_FWD_COMM
      ANB
      ORB
      LD      D7554.0  ; NST6_SEALING_UNIT3_MOVE_COND
      OR      D7552.0  ; NST6_SEALING_UNIT3_FWD_COMM
      ANB
      ANI     D7552.1  ; NST6_SEALING_UNIT3_RET_COMM
      ANI     D7559.7  ; NST6_SEALING_UNIT3_EMERG_RET_COM
      OUT     D7552.0  ; NST6_SEALING_UNIT3_FWD_COMM
; Rung 151
1742  LD      D7500.6  ; NST6_ALL_CYCLE_CMPLT1
      OR      D7559.7  ; NST6_SEALING_UNIT3_EMERG_RET_COM
      AND     D5000.0  ; CKT2_AUTO_COTROL
      LDI     D7550.0  ; NST6_SEALING_UNIT3_BACK
      AND     L1594  ; NST6 MAN REV BTN
      ANI     L1593  ; NST6 MAN FWD BTN
      AND     D7506.2  ; NST6_SEALING_UNIT_THREE_SELECT
      ORB
      ANI     D7552.0  ; NST6_SEALING_UNIT3_FWD_COMM
      ANI     D7550.0  ; NST6_SEALING_UNIT3_BACK
      OUT     D7552.1  ; NST6_SEALING_UNIT3_RET_COMM
; Rung 152
1759  LD      D7552.0  ; NST6_SEALING_UNIT3_FWD_COMM
      SET     D7552.2  ; NST6_SEALING_UNIT3_FWD_COMM_RETA
; Rung 153
1767  LD      D7552.1  ; NST6_SEALING_UNIT3_RET_COMM
      SET     D7552.3  ; NST6_SEALING_UNIT3_RET_COMM_RETA
; Rung 154
1775  LD      D7552.1  ; NST6_SEALING_UNIT3_RET_COMM
      OR      D7552.3  ; NST6_SEALING_UNIT3_RET_COMM_RETA
      RST     D7552.2  ; NST6_SEALING_UNIT3_FWD_COMM_RETA
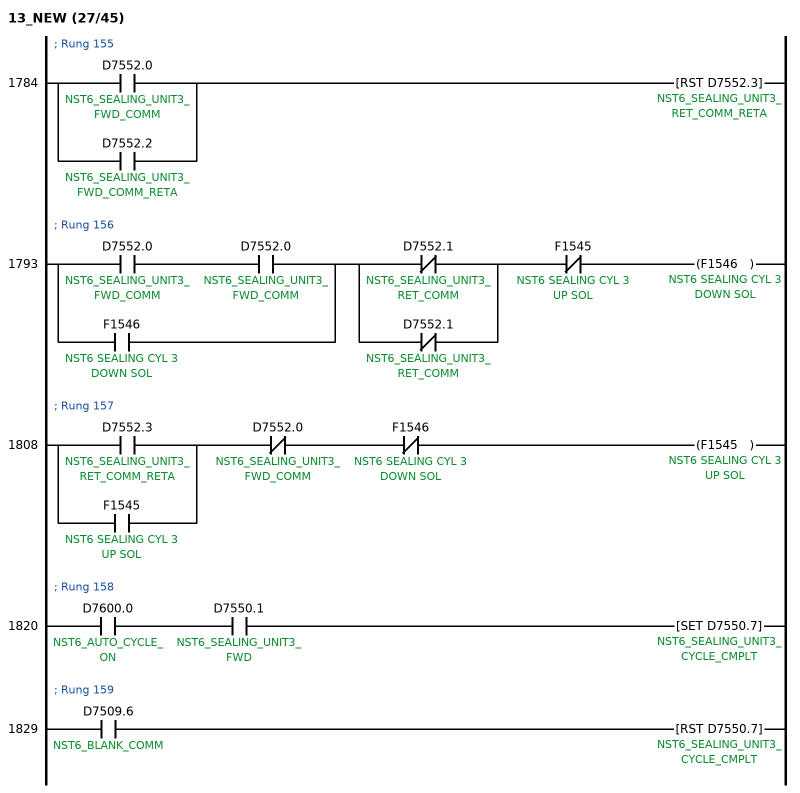
; Rung 155
1784  LD      D7552.0  ; NST6_SEALING_UNIT3_FWD_COMM
      OR      D7552.2  ; NST6_SEALING_UNIT3_FWD_COMM_RETA
      RST     D7552.3  ; NST6_SEALING_UNIT3_RET_COMM_RETA
; Rung 156
1793  LD      D7552.0  ; NST6_SEALING_UNIT3_FWD_COMM
      AND     D7552.0  ; NST6_SEALING_UNIT3_FWD_COMM
      OR      F1546  ; NST6 SEALING CYL 3 DOWN SOL
      LDI     D7552.1  ; NST6_SEALING_UNIT3_RET_COMM
      ORI     D7552.1  ; NST6_SEALING_UNIT3_RET_COMM
      ANB
      ANI     F1545  ; NST6 SEALING CYL 3 UP SOL
      OUT     F1546  ; NST6 SEALING CYL 3 DOWN SOL
; Rung 157
1808  LD      D7552.3  ; NST6_SEALING_UNIT3_RET_COMM_RETA
      OR      F1545  ; NST6 SEALING CYL 3 UP SOL
      ANI     D7552.0  ; NST6_SEALING_UNIT3_FWD_COMM
      ANI     F1546  ; NST6 SEALING CYL 3 DOWN SOL
      OUT     F1545  ; NST6 SEALING CYL 3 UP SOL
; Rung 158
1820  LD      D7600.0  ; NST6_AUTO_CYCLE_ON
      AND     D7550.1  ; NST6_SEALING_UNIT3_FWD
      SET     D7550.7  ; NST6_SEALING_UNIT3_CYCLE_CMPLT
; Rung 159
1829  LD      D7509.6  ; NST6_BLANK_COMM
      RST     D7550.7  ; NST6_SEALING_UNIT3_CYCLE_CMPLT
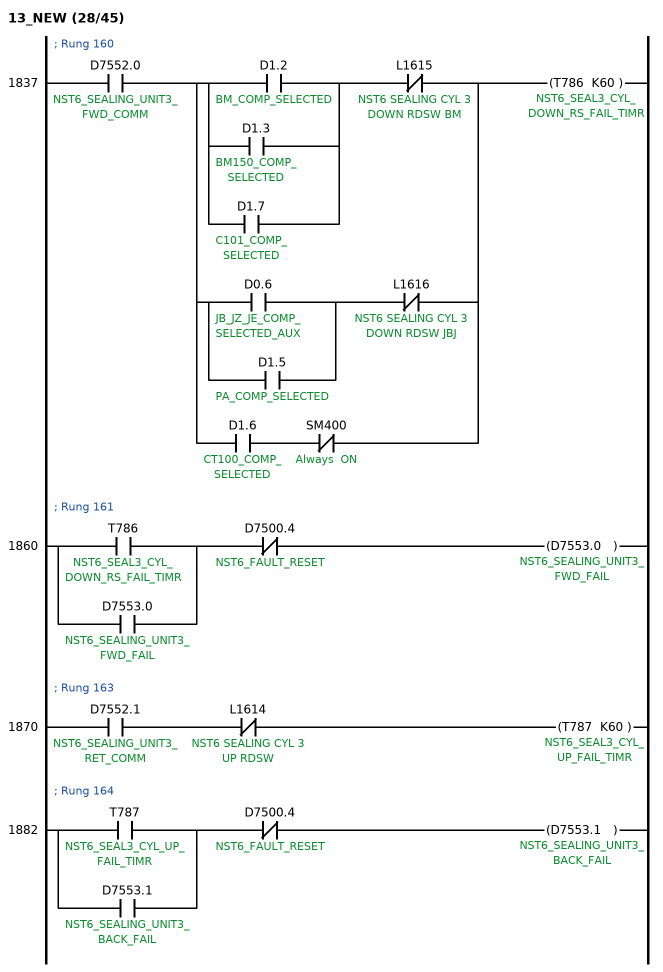
; Rung 160
1837  LD      D7552.0  ; NST6_SEALING_UNIT3_FWD_COMM
      LD      D1.2  ; BM_COMP_SELECTED
      OR      D1.3  ; BM150_COMP_SELECTED
      OR      D1.7  ; C101_COMP_SELECTED
      ANI     L1615  ; NST6 SEALING CYL 3 DOWN RDSW BM
      LD      D0.6  ; JB_JZ_JE_COMP_SELECTED_AUX
      OR      D1.5  ; PA_COMP_SELECTED
      ANI     L1616  ; NST6 SEALING CYL 3 DOWN RDSW JBJ
      ORB
      LD      D1.6  ; CT100_COMP_SELECTED
      ANI     SM400  ; Always  ON
      ORB
      ANB
      OUT     T786 K60  ; NST6_SEAL3_CYL_DOWN_RS_FAIL_TIMR
; Rung 161
1860  LD      T786  ; NST6_SEAL3_CYL_DOWN_RS_FAIL_TIMR
      OR      D7553.0  ; NST6_SEALING_UNIT3_FWD_FAIL
      ANI     D7500.4  ; NST6_FAULT_RESET
      OUT     D7553.0  ; NST6_SEALING_UNIT3_FWD_FAIL
; Rung 163
1870  LD      D7552.1  ; NST6_SEALING_UNIT3_RET_COMM
      ANI     L1614  ; NST6 SEALING CYL 3 UP RDSW
      OUT     T787 K60  ; NST6_SEAL3_CYL_UP_FAIL_TIMR
; Rung 164
1882  LD      T787  ; NST6_SEAL3_CYL_UP_FAIL_TIMR
      OR      D7553.1  ; NST6_SEALING_UNIT3_BACK_FAIL
      ANI     D7500.4  ; NST6_FAULT_RESET
      OUT     D7553.1  ; NST6_SEALING_UNIT3_BACK_FAIL
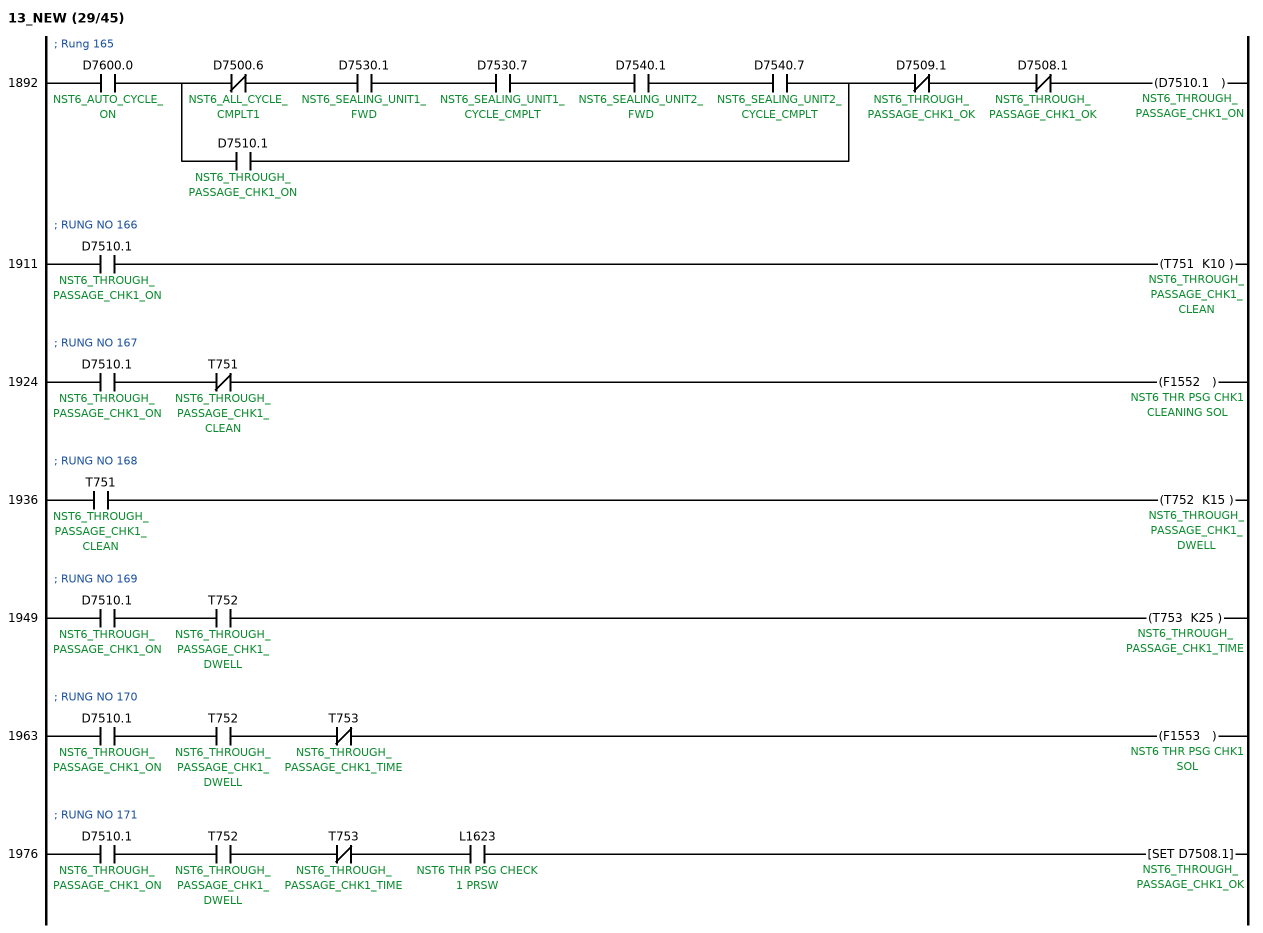
; Rung 165
1892  LD      D7600.0  ; NST6_AUTO_CYCLE_ON
      LDI     D7500.6  ; NST6_ALL_CYCLE_CMPLT1
      AND     D7530.1  ; NST6_SEALING_UNIT1_FWD
      AND     D7530.7  ; NST6_SEALING_UNIT1_CYCLE_CMPLT
      AND     D7540.1  ; NST6_SEALING_UNIT2_FWD
      AND     D7540.7  ; NST6_SEALING_UNIT2_CYCLE_CMPLT
      OR      D7510.1  ; NST6_THROUGH_PASSAGE_CHK1_ON
      ANB
      ANI     D7509.1  ; NST6_THROUGH_PASSAGE_CHK1_OK
      ANI     D7508.1  ; NST6_THROUGH_PASSAGE_CHK1_OK
      OUT     D7510.1  ; NST6_THROUGH_PASSAGE_CHK1_ON
; RUNG NO 166
1911  LD      D7510.1  ; NST6_THROUGH_PASSAGE_CHK1_ON
      OUT     T751 K10  ; NST6_THROUGH_PASSAGE_CHK1_CLEAN
; RUNG NO 167
1924  LD      D7510.1  ; NST6_THROUGH_PASSAGE_CHK1_ON
      ANI     T751  ; NST6_THROUGH_PASSAGE_CHK1_CLEAN
      OUT     F1552  ; NST6 THR PSG CHK1 CLEANING SOL
; RUNG NO 168
1936  LD      T751  ; NST6_THROUGH_PASSAGE_CHK1_CLEAN
      OUT     T752 K15  ; NST6_THROUGH_PASSAGE_CHK1_DWELL
; RUNG NO 169
1949  LD      D7510.1  ; NST6_THROUGH_PASSAGE_CHK1_ON
      AND     T752  ; NST6_THROUGH_PASSAGE_CHK1_DWELL
      OUT     T753 K25  ; NST6_THROUGH_PASSAGE_CHK1_TIME
; RUNG NO 170
1963  LD      D7510.1  ; NST6_THROUGH_PASSAGE_CHK1_ON
      AND     T752  ; NST6_THROUGH_PASSAGE_CHK1_DWELL
      ANI     T753  ; NST6_THROUGH_PASSAGE_CHK1_TIME
      OUT     F1553  ; NST6 THR PSG CHK1 SOL
; RUNG NO 171
1976  LD      D7510.1  ; NST6_THROUGH_PASSAGE_CHK1_ON
      AND     T752  ; NST6_THROUGH_PASSAGE_CHK1_DWELL
      ANI     T753  ; NST6_THROUGH_PASSAGE_CHK1_TIME
      AND     L1623  ; NST6 THR PSG CHECK 1 PRSW
      SET     D7508.1  ; NST6_THROUGH_PASSAGE_CHK1_OK
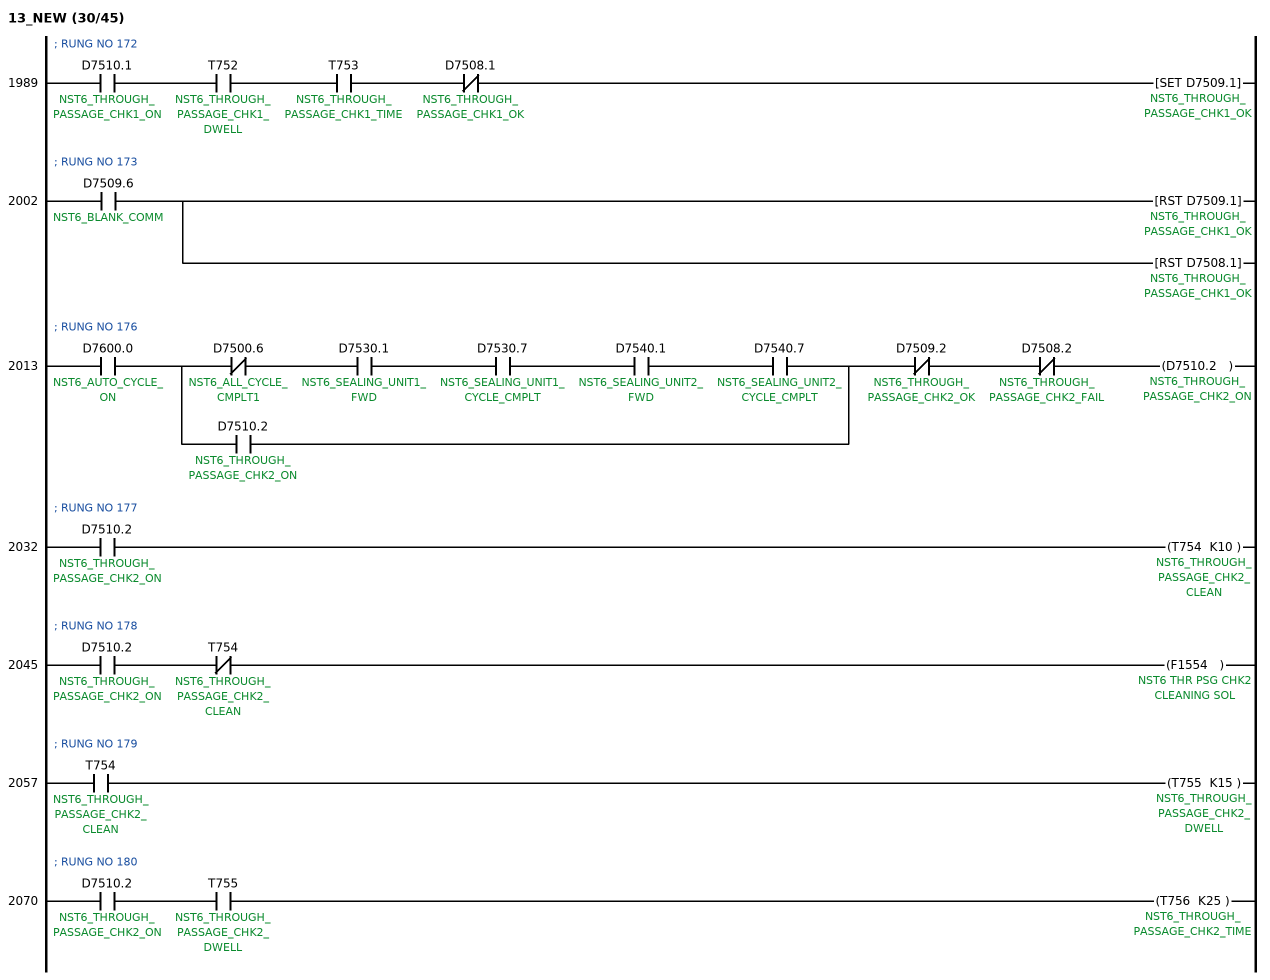
; RUNG NO 172
1989  LD      D7510.1  ; NST6_THROUGH_PASSAGE_CHK1_ON
      AND     T752  ; NST6_THROUGH_PASSAGE_CHK1_DWELL
      AND     T753  ; NST6_THROUGH_PASSAGE_CHK1_TIME
      ANI     D7508.1  ; NST6_THROUGH_PASSAGE_CHK1_OK
      SET     D7509.1  ; NST6_THROUGH_PASSAGE_CHK1_OK
; RUNG NO 173
2002  LD      D7509.6  ; NST6_BLANK_COMM
      RST     D7509.1  ; NST6_THROUGH_PASSAGE_CHK1_OK
      RST     D7508.1  ; NST6_THROUGH_PASSAGE_CHK1_OK
; RUNG NO 176
2013  LD      D7600.0  ; NST6_AUTO_CYCLE_ON
      LDI     D7500.6  ; NST6_ALL_CYCLE_CMPLT1
      AND     D7530.1  ; NST6_SEALING_UNIT1_FWD
      AND     D7530.7  ; NST6_SEALING_UNIT1_CYCLE_CMPLT
      AND     D7540.1  ; NST6_SEALING_UNIT2_FWD
      AND     D7540.7  ; NST6_SEALING_UNIT2_CYCLE_CMPLT
      OR      D7510.2  ; NST6_THROUGH_PASSAGE_CHK2_ON
      ANB
      ANI     D7509.2  ; NST6_THROUGH_PASSAGE_CHK2_OK
      ANI     D7508.2  ; NST6_THROUGH_PASSAGE_CHK2_FAIL
      OUT     D7510.2  ; NST6_THROUGH_PASSAGE_CHK2_ON
; RUNG NO 177
2032  LD      D7510.2  ; NST6_THROUGH_PASSAGE_CHK2_ON
      OUT     T754 K10  ; NST6_THROUGH_PASSAGE_CHK2_CLEAN
; RUNG NO 178
2045  LD      D7510.2  ; NST6_THROUGH_PASSAGE_CHK2_ON
      ANI     T754  ; NST6_THROUGH_PASSAGE_CHK2_CLEAN
      OUT     F1554  ; NST6 THR PSG CHK2 CLEANING SOL
; RUNG NO 179
2057  LD      T754  ; NST6_THROUGH_PASSAGE_CHK2_CLEAN
      OUT     T755 K15  ; NST6_THROUGH_PASSAGE_CHK2_DWELL
; RUNG NO 180
2070  LD      D7510.2  ; NST6_THROUGH_PASSAGE_CHK2_ON
      AND     T755  ; NST6_THROUGH_PASSAGE_CHK2_DWELL
      OUT     T756 K25  ; NST6_THROUGH_PASSAGE_CHK2_TIME
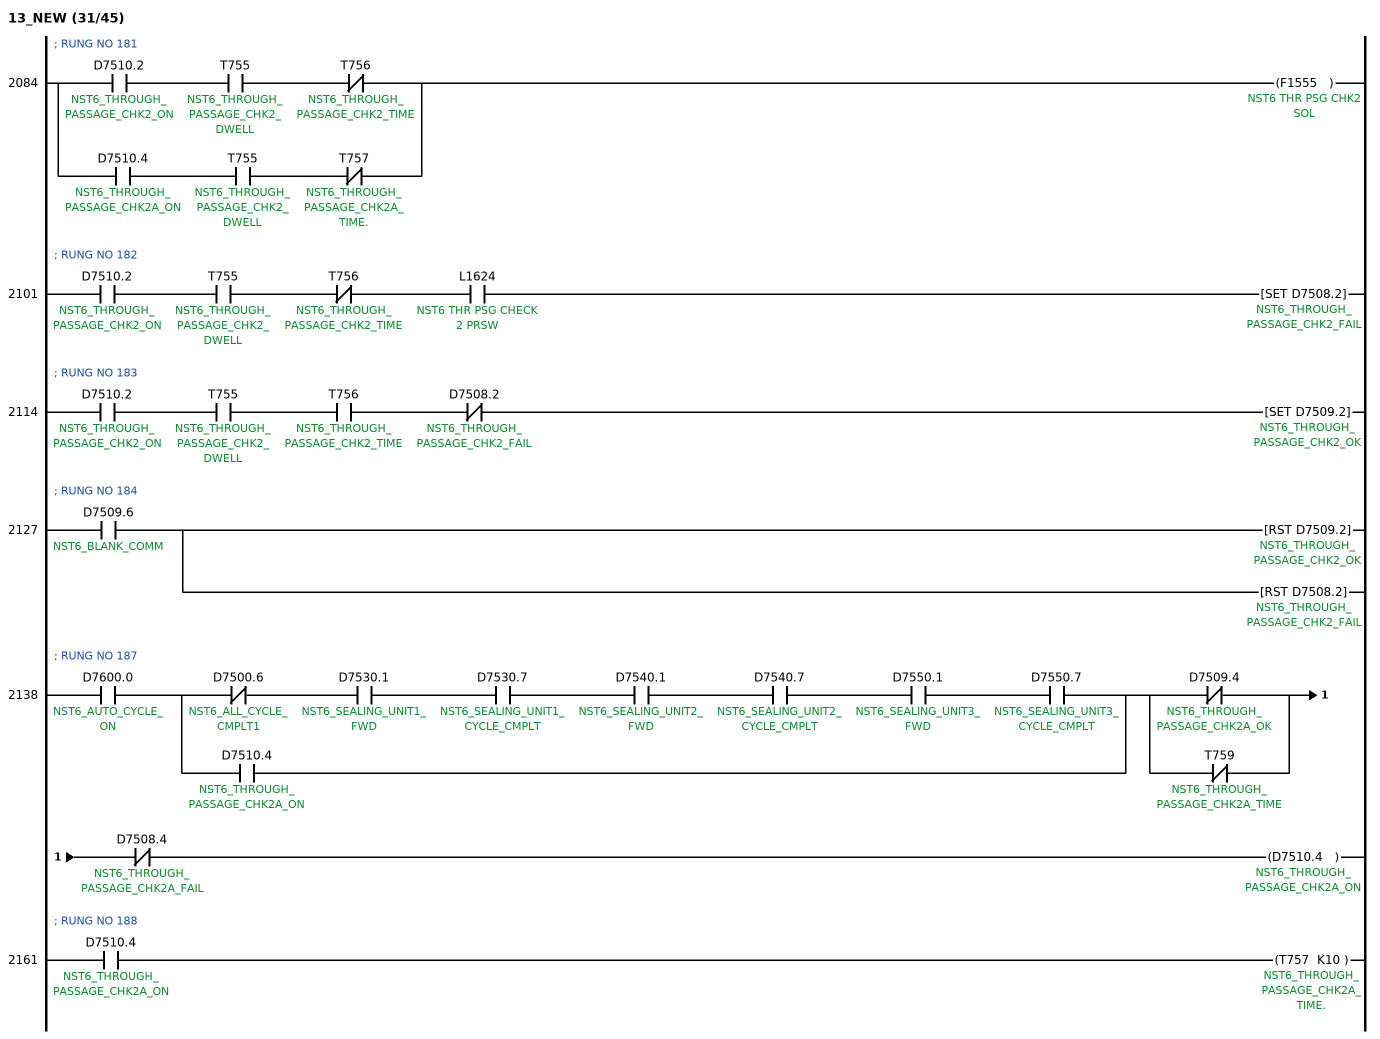
; RUNG NO 181
2084  LD      D7510.2  ; NST6_THROUGH_PASSAGE_CHK2_ON
      AND     T755  ; NST6_THROUGH_PASSAGE_CHK2_DWELL
      ANI     T756  ; NST6_THROUGH_PASSAGE_CHK2_TIME
      LD      D7510.4  ; NST6_THROUGH_PASSAGE_CHK2A_ON
      AND     T755  ; NST6_THROUGH_PASSAGE_CHK2_DWELL
      ANI     T757  ; NST6_THROUGH_PASSAGE_CHK2A_TIME.
      ORB
      OUT     F1555  ; NST6 THR PSG CHK2 SOL
; RUNG NO 182
2101  LD      D7510.2  ; NST6_THROUGH_PASSAGE_CHK2_ON
      AND     T755  ; NST6_THROUGH_PASSAGE_CHK2_DWELL
      ANI     T756  ; NST6_THROUGH_PASSAGE_CHK2_TIME
      AND     L1624  ; NST6 THR PSG CHECK 2 PRSW
      SET     D7508.2  ; NST6_THROUGH_PASSAGE_CHK2_FAIL
; RUNG NO 183
2114  LD      D7510.2  ; NST6_THROUGH_PASSAGE_CHK2_ON
      AND     T755  ; NST6_THROUGH_PASSAGE_CHK2_DWELL
      AND     T756  ; NST6_THROUGH_PASSAGE_CHK2_TIME
      ANI     D7508.2  ; NST6_THROUGH_PASSAGE_CHK2_FAIL
      SET     D7509.2  ; NST6_THROUGH_PASSAGE_CHK2_OK
; RUNG NO 184
2127  LD      D7509.6  ; NST6_BLANK_COMM
      RST     D7509.2  ; NST6_THROUGH_PASSAGE_CHK2_OK
      RST     D7508.2  ; NST6_THROUGH_PASSAGE_CHK2_FAIL
; RUNG NO 187
2138  LD      D7600.0  ; NST6_AUTO_CYCLE_ON
      LDI     D7500.6  ; NST6_ALL_CYCLE_CMPLT1
      AND     D7530.1  ; NST6_SEALING_UNIT1_FWD
      AND     D7530.7  ; NST6_SEALING_UNIT1_CYCLE_CMPLT
      AND     D7540.1  ; NST6_SEALING_UNIT2_FWD
      AND     D7540.7  ; NST6_SEALING_UNIT2_CYCLE_CMPLT
      AND     D7550.1  ; NST6_SEALING_UNIT3_FWD
      AND     D7550.7  ; NST6_SEALING_UNIT3_CYCLE_CMPLT
      OR      D7510.4  ; NST6_THROUGH_PASSAGE_CHK2A_ON
      ANB
      LDI     D7509.4  ; NST6_THROUGH_PASSAGE_CHK2A_OK
      ORI     T759  ; NST6_THROUGH_PASSAGE_CHK2A_TIME
      ANB
      ANI     D7508.4  ; NST6_THROUGH_PASSAGE_CHK2A_FAIL
      OUT     D7510.4  ; NST6_THROUGH_PASSAGE_CHK2A_ON
; RUNG NO 188
2161  LD      D7510.4  ; NST6_THROUGH_PASSAGE_CHK2A_ON
      OUT     T757 K10  ; NST6_THROUGH_PASSAGE_CHK2A_TIME.
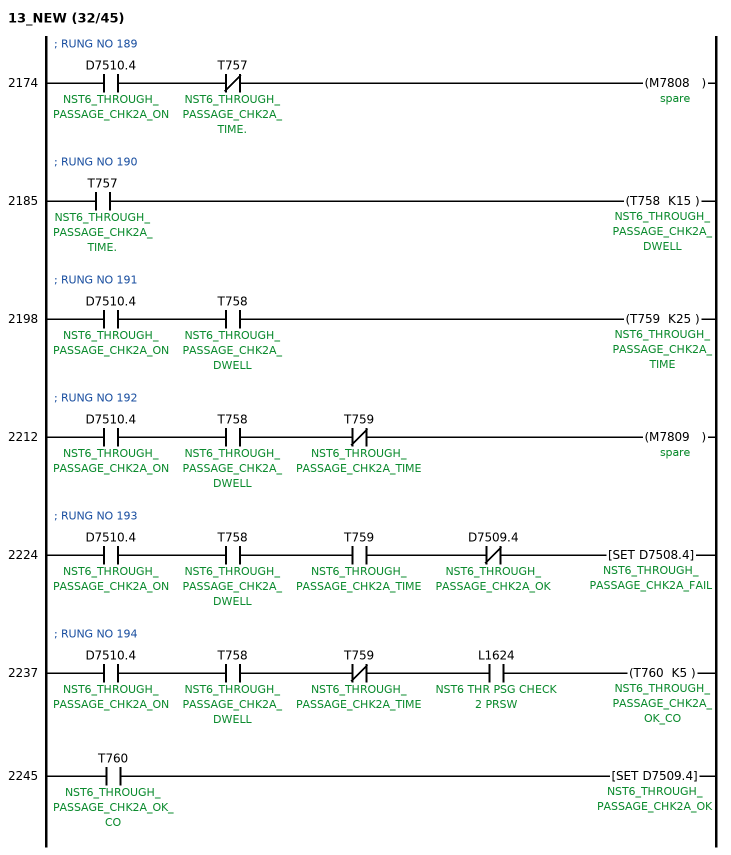
; RUNG NO 189
2174  LD      D7510.4  ; NST6_THROUGH_PASSAGE_CHK2A_ON
      ANI     T757  ; NST6_THROUGH_PASSAGE_CHK2A_TIME.
      OUT     M7808  ; spare
; RUNG NO 190
2185  LD      T757  ; NST6_THROUGH_PASSAGE_CHK2A_TIME.
      OUT     T758 K15  ; NST6_THROUGH_PASSAGE_CHK2A_DWELL
; RUNG NO 191
2198  LD      D7510.4  ; NST6_THROUGH_PASSAGE_CHK2A_ON
      AND     T758  ; NST6_THROUGH_PASSAGE_CHK2A_DWELL
      OUT     T759 K25  ; NST6_THROUGH_PASSAGE_CHK2A_TIME
; RUNG NO 192
2212  LD      D7510.4  ; NST6_THROUGH_PASSAGE_CHK2A_ON
      AND     T758  ; NST6_THROUGH_PASSAGE_CHK2A_DWELL
      ANI     T759  ; NST6_THROUGH_PASSAGE_CHK2A_TIME
      OUT     M7809  ; spare
; RUNG NO 193
2224  LD      D7510.4  ; NST6_THROUGH_PASSAGE_CHK2A_ON
      AND     T758  ; NST6_THROUGH_PASSAGE_CHK2A_DWELL
      AND     T759  ; NST6_THROUGH_PASSAGE_CHK2A_TIME
      ANI     D7509.4  ; NST6_THROUGH_PASSAGE_CHK2A_OK
      SET     D7508.4  ; NST6_THROUGH_PASSAGE_CHK2A_FAIL
; RUNG NO 194
2237  LD      D7510.4  ; NST6_THROUGH_PASSAGE_CHK2A_ON
      AND     T758  ; NST6_THROUGH_PASSAGE_CHK2A_DWELL
      ANI     T759  ; NST6_THROUGH_PASSAGE_CHK2A_TIME
      AND     L1624  ; NST6 THR PSG CHECK 2 PRSW
      OUT     T760 K5  ; NST6_THROUGH_PASSAGE_CHK2A_OK_CO
2245  LD      T760  ; NST6_THROUGH_PASSAGE_CHK2A_OK_CO
      SET     D7509.4  ; NST6_THROUGH_PASSAGE_CHK2A_OK
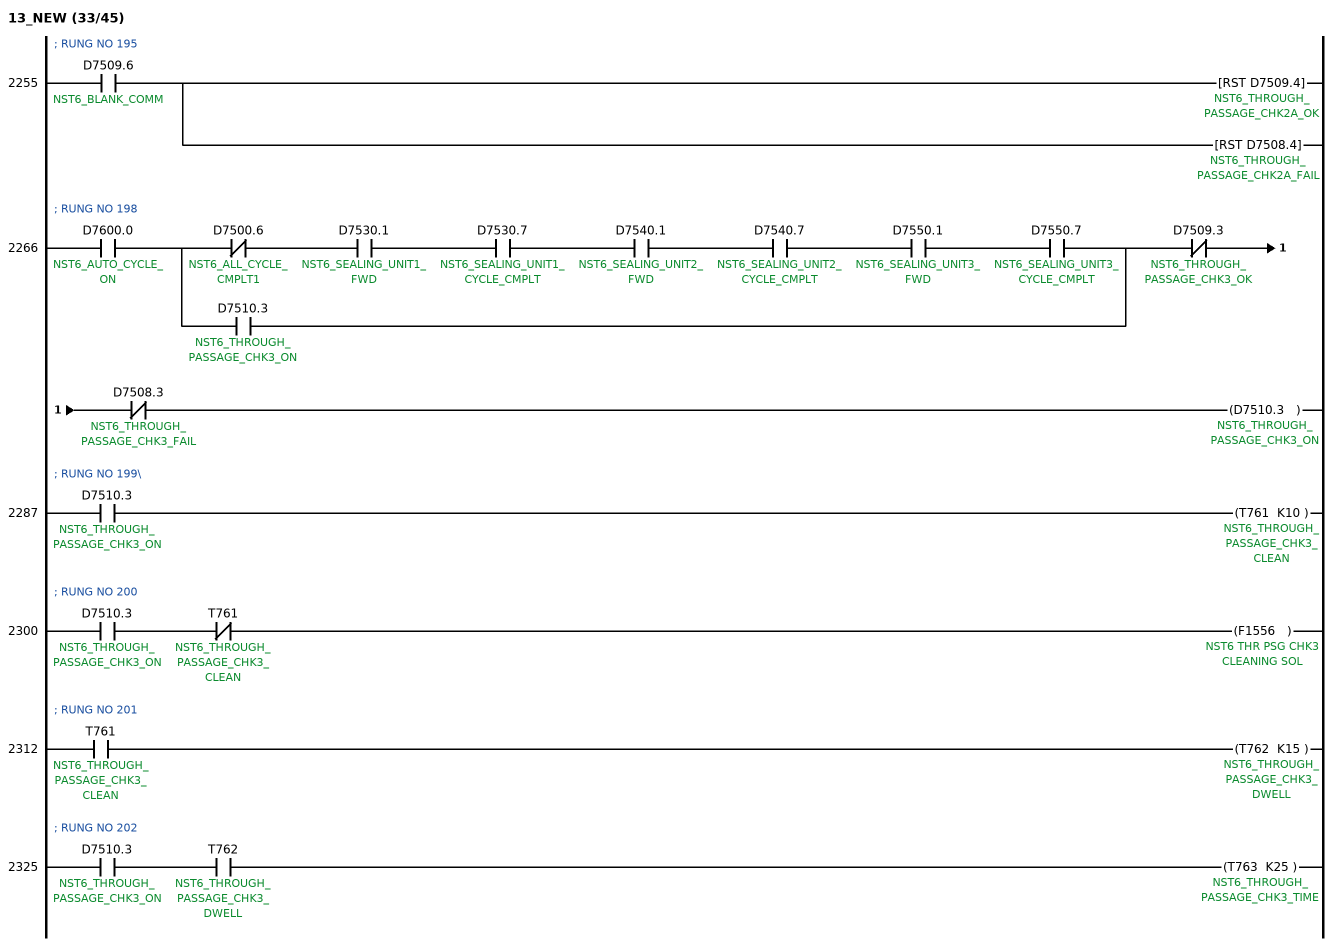
; RUNG NO 195
2255  LD      D7509.6  ; NST6_BLANK_COMM
      RST     D7509.4  ; NST6_THROUGH_PASSAGE_CHK2A_OK
      RST     D7508.4  ; NST6_THROUGH_PASSAGE_CHK2A_FAIL
; RUNG NO 198
2266  LD      D7600.0  ; NST6_AUTO_CYCLE_ON
      LDI     D7500.6  ; NST6_ALL_CYCLE_CMPLT1
      AND     D7530.1  ; NST6_SEALING_UNIT1_FWD
      AND     D7530.7  ; NST6_SEALING_UNIT1_CYCLE_CMPLT
      AND     D7540.1  ; NST6_SEALING_UNIT2_FWD
      AND     D7540.7  ; NST6_SEALING_UNIT2_CYCLE_CMPLT
      AND     D7550.1  ; NST6_SEALING_UNIT3_FWD
      AND     D7550.7  ; NST6_SEALING_UNIT3_CYCLE_CMPLT
      OR      D7510.3  ; NST6_THROUGH_PASSAGE_CHK3_ON
      ANB
      ANI     D7509.3  ; NST6_THROUGH_PASSAGE_CHK3_OK
      ANI     D7508.3  ; NST6_THROUGH_PASSAGE_CHK3_FAIL
      OUT     D7510.3  ; NST6_THROUGH_PASSAGE_CHK3_ON
; RUNG NO 199\
2287  LD      D7510.3  ; NST6_THROUGH_PASSAGE_CHK3_ON
      OUT     T761 K10  ; NST6_THROUGH_PASSAGE_CHK3_CLEAN
; RUNG NO 200
2300  LD      D7510.3  ; NST6_THROUGH_PASSAGE_CHK3_ON
      ANI     T761  ; NST6_THROUGH_PASSAGE_CHK3_CLEAN
      OUT     F1556  ; NST6 THR PSG CHK3 CLEANING SOL
; RUNG NO 201
2312  LD      T761  ; NST6_THROUGH_PASSAGE_CHK3_CLEAN
      OUT     T762 K15  ; NST6_THROUGH_PASSAGE_CHK3_DWELL
; RUNG NO 202
2325  LD      D7510.3  ; NST6_THROUGH_PASSAGE_CHK3_ON
      AND     T762  ; NST6_THROUGH_PASSAGE_CHK3_DWELL
      OUT     T763 K25  ; NST6_THROUGH_PASSAGE_CHK3_TIME
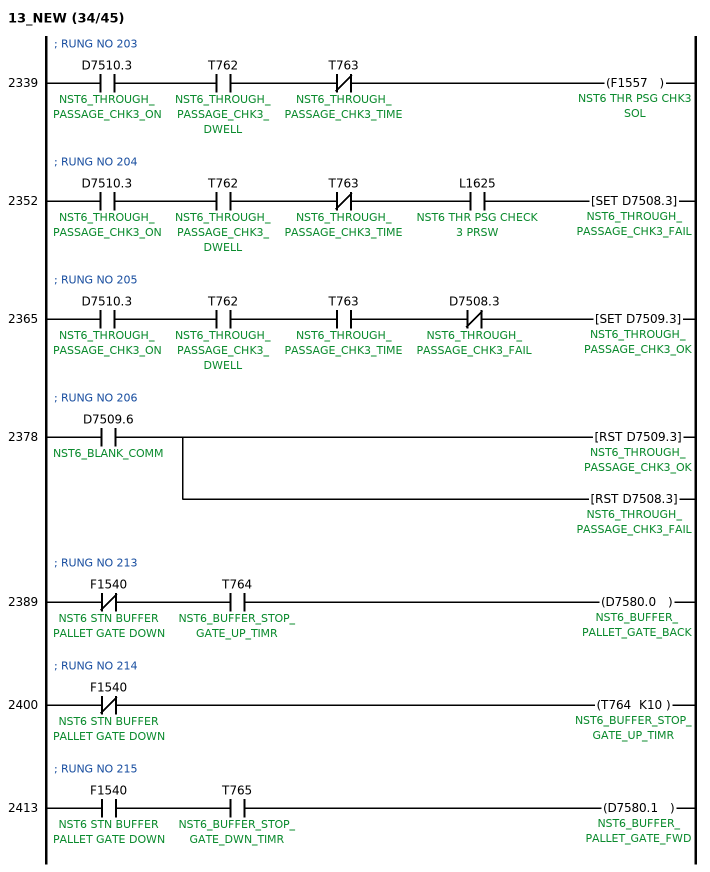
; RUNG NO 203
2339  LD      D7510.3  ; NST6_THROUGH_PASSAGE_CHK3_ON
      AND     T762  ; NST6_THROUGH_PASSAGE_CHK3_DWELL
      ANI     T763  ; NST6_THROUGH_PASSAGE_CHK3_TIME
      OUT     F1557  ; NST6 THR PSG CHK3 SOL
; RUNG NO 204
2352  LD      D7510.3  ; NST6_THROUGH_PASSAGE_CHK3_ON
      AND     T762  ; NST6_THROUGH_PASSAGE_CHK3_DWELL
      ANI     T763  ; NST6_THROUGH_PASSAGE_CHK3_TIME
      AND     L1625  ; NST6 THR PSG CHECK 3 PRSW
      SET     D7508.3  ; NST6_THROUGH_PASSAGE_CHK3_FAIL
; RUNG NO 205
2365  LD      D7510.3  ; NST6_THROUGH_PASSAGE_CHK3_ON
      AND     T762  ; NST6_THROUGH_PASSAGE_CHK3_DWELL
      AND     T763  ; NST6_THROUGH_PASSAGE_CHK3_TIME
      ANI     D7508.3  ; NST6_THROUGH_PASSAGE_CHK3_FAIL
      SET     D7509.3  ; NST6_THROUGH_PASSAGE_CHK3_OK
; RUNG NO 206
2378  LD      D7509.6  ; NST6_BLANK_COMM
      RST     D7509.3  ; NST6_THROUGH_PASSAGE_CHK3_OK
      RST     D7508.3  ; NST6_THROUGH_PASSAGE_CHK3_FAIL
; RUNG NO 213
2389  LDI     F1540  ; NST6 STN BUFFER PALLET GATE DOWN
      AND     T764  ; NST6_BUFFER_STOP_GATE_UP_TIMR
      OUT     D7580.0  ; NST6_BUFFER_PALLET_GATE_BACK
; RUNG NO 214
2400  LDI     F1540  ; NST6 STN BUFFER PALLET GATE DOWN
      OUT     T764 K10  ; NST6_BUFFER_STOP_GATE_UP_TIMR
; RUNG NO 215
2413  LD      F1540  ; NST6 STN BUFFER PALLET GATE DOWN
      AND     T765  ; NST6_BUFFER_STOP_GATE_DWN_TIMR
      OUT     D7580.1  ; NST6_BUFFER_PALLET_GATE_FWD
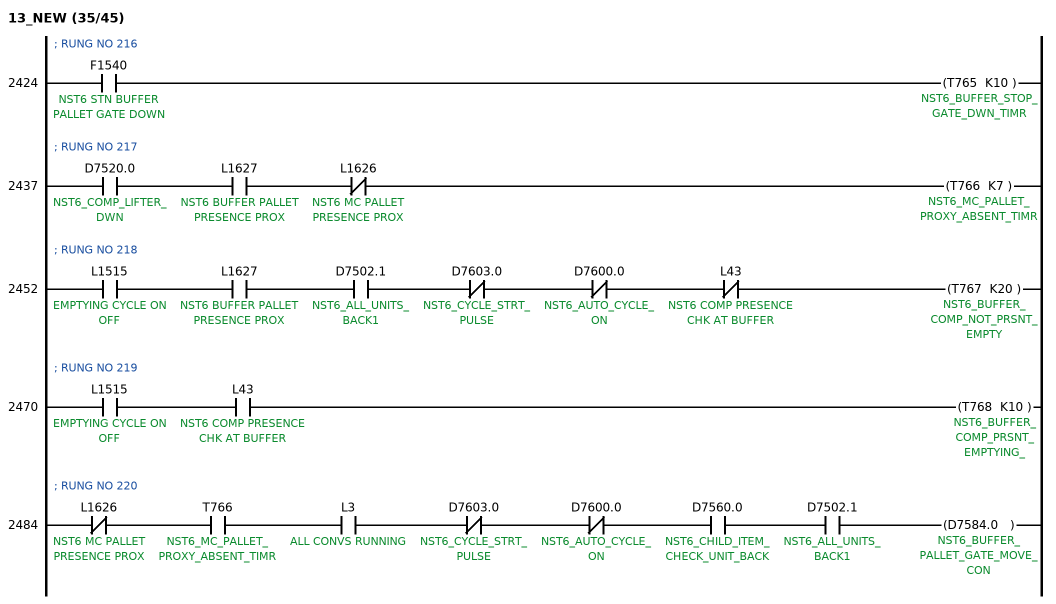
; RUNG NO 216
2424  LD      F1540  ; NST6 STN BUFFER PALLET GATE DOWN
      OUT     T765 K10  ; NST6_BUFFER_STOP_GATE_DWN_TIMR
; RUNG NO 217
2437  LD      D7520.0  ; NST6_COMP_LIFTER_DWN
      AND     L1627  ; NST6 BUFFER PALLET PRESENCE PROX
      ANI     L1626  ; NST6 MC PALLET PRESENCE PROX
      OUT     T766 K7  ; NST6_MC_PALLET_PROXY_ABSENT_TIMR
; RUNG NO 218
2452  LD      L1515  ; EMPTYING CYCLE ON OFF
      AND     L1627  ; NST6 BUFFER PALLET PRESENCE PROX
      AND     D7502.1  ; NST6_ALL_UNITS_BACK1
      ANI     D7603.0  ; NST6_CYCLE_STRT_PULSE
      ANI     D7600.0  ; NST6_AUTO_CYCLE_ON
      ANI     L43  ; NST6 COMP PRESENCE CHK AT BUFFER
      OUT     T767 K20  ; NST6_BUFFER_COMP_NOT_PRSNT_EMPTY
; RUNG NO 219
2470  LD      L1515  ; EMPTYING CYCLE ON OFF
      AND     L43  ; NST6 COMP PRESENCE CHK AT BUFFER
      OUT     T768 K10  ; NST6_BUFFER_COMP_PRSNT_EMPTYING_
; RUNG NO 220
2484  LDI     L1626  ; NST6 MC PALLET PRESENCE PROX
      AND     T766  ; NST6_MC_PALLET_PROXY_ABSENT_TIMR
      AND     L3  ; ALL CONVS RUNNING
      ANI     D7603.0  ; NST6_CYCLE_STRT_PULSE
      ANI     D7600.0  ; NST6_AUTO_CYCLE_ON
      AND     D7560.0  ; NST6_CHILD_ITEM_CHECK_UNIT_BACK
      AND     D7502.1  ; NST6_ALL_UNITS_BACK1
      OUT     D7584.0  ; NST6_BUFFER_PALLET_GATE_MOVE_CON
